KUKA KRL program: MyProgram_168().src

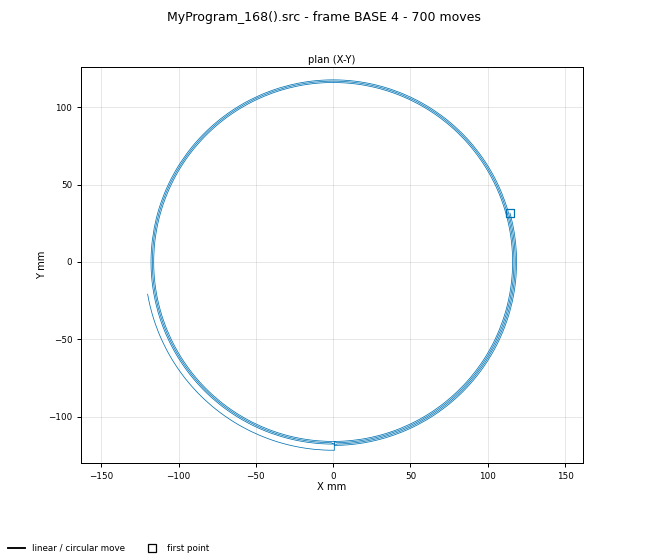
[picture p0: tool path of MyProgram_168().src in frame BASE 4, 700 of 700 moves have a stored position in this frame; points joined in program order, loops and branches not executed]
&ACCESS RVP
&REL 1
&PARAM TEMPLATE = C:\KRC\Roboter\Template\vorgabe
&PARAM EDITMASK = *
DEF MyProgram_168()
; ---- Setting reference (Base) ----
$BASE = BASE_DATA[4]

; --------------------------
; ---- Setting tool (TCP) ----
$TOOL = TOOL_DATA[3]
; --------------------------

$VEL.CP = VEL_APROX_PRINT
Startdeposition()
$VEL.CP = VEL_PRINT
LIN {X 114.3697,Y 31.6504,Z 126,A 10.9682,B 24.9468,C -1.6846,E1 25.1544,E2 435.1117} C_DIS
LIN {X 115.2864,Y 28.1194,Z 126,A 9.3071,B 24.9468,C -1.6839,E1 25.1555,E2 436.7647} C_DIS
LIN {X 116.1642,Y 24.242,Z 126,A 7.4646,B 24.947,C -1.6816,E1 25.1566,E2 438.602} C_DIS
LIN {X 116.7128,Y 21.447,Z 126,A 6.0097,B 24.9475,C -1.6734,E1 25.1574,E2 440.0678} C_DIS
LIN {X 117.2786,Y 18.0937,Z 126,A 4.4449,B 24.9476,C -1.6719,E1 25.1581,E2 441.6268} C_DIS
LIN {X 117.7204,Y 14.9551,Z 126,A 2.982,B 24.9477,C -1.6702,E1 25.1586,E2 443.0851} C_DIS
LIN {X 118.1031,Y 11.5648,Z 126,A 1.1366,B 24.9487,C -1.6553,E1 25.1592,E2 444.9547} C_DIS
LIN {X 118.5333,Y 5.6393,Z 126,A -1.9787,B 24.95,C -1.6341,E1 25.1597,E2 448.1015} C_DIS
LIN {X 118.6444,Y 2.2744,Z 126,A -3.2425,B 24.9492,C -1.6463,E1 25.1597,E2 449.3291} C_DIS
LIN {X 118.6544,Y -1.7308,Z 126,A -5.1222,B 24.9494,C -1.6426,E1 25.1597,E2 451.2063} C_DIS
LIN {X 118.3168,Y -9.105,Z 126,A -8.6006,B 24.9499,C -1.635,E1 25.1593,E2 454.6818} C_DIS
LIN {X 118.0451,Y -12.1269,Z 126,A -10.0562,B 24.9502,C -1.6307,E1 25.1589,E2 456.139} C_DIS
LIN {X 117.691,Y -15.182,Z 126,A -11.6024,B 24.9506,C -1.6229,E1 25.1583,E2 457.6945} C_DIS
LIN {X 117.1469,Y -18.9382,Z 126,A -13.4854,B 24.9512,C -1.6144,E1 25.1575,E2 459.5865} C_DIS
LIN {X 116.5226,Y -22.453,Z 126,A -15.1525,B 24.9513,C -1.6116,E1 25.1567,E2 461.2505} C_DIS
LIN {X 115.7438,Y -26.1788,Z 126,A -16.9413,B 24.9516,C -1.608,E1 25.1556,E2 463.0374} C_DIS
LIN {X 114.3078,Y -31.8689,Z 126,A -19.8139,B 24.9522,C -1.5969,E1 25.1536,E2 465.9193} C_DIS
LIN {X 113.3954,Y -34.9736,Z 126,A -21.3368,B 24.9524,C -1.5939,E1 25.1524,E2 467.4408} C_DIS
LIN {X 112.2692,Y -38.4394,Z 126,A -23.1908,B 24.953,C -1.5837,E1 25.1507,E2 469.3084} C_DIS
LIN {X 110.9509,Y -42.0898,Z 126,A -24.8724,B 24.9528,C -1.5872,E1 25.1491,E2 470.9724} C_DIS
LIN {X 109.7246,Y -45.1929,Z 126,A -27.2104,B 24.9552,C -1.5471,E1 25.1466,E2 473.392} C_DIS
LIN {X 107.7996,Y -49.6101,Z 126,A -28.9531,B 24.9539,C -1.568,E1 25.1446,E2 475.0759} C_DIS
LIN {X 105.9977,Y -53.3542,Z 126,A -30.9386,B 24.9542,C -1.5629,E1 25.1422,E2 477.0628} C_DIS
LIN {X 104.0576,Y -57.0433,Z 126,A -33.1637,B 24.9552,C -1.5467,E1 25.1392,E2 479.3145} C_DIS
LIN {X 102.4696,Y -59.8499,Z 126,A -34.2864,B 24.9542,C -1.563,E1 25.1377,E2 480.3929} C_DIS
LIN {X 99.8547,Y -64.1146,Z 126,A -36.7516,B 24.9548,C -1.5536,E1 25.134,E2 482.8677} C_DIS
LIN {X 96.6923,Y -68.7916,Z 126,A -39.4176,B 24.9551,C -1.5488,E1 25.1298,E2 485.5319} C_DIS
LIN {X 95.1595,Y -70.898,Z 126,A -40.5832,B 24.9551,C -1.5497,E1 25.1279,E2 486.6897} C_DIS
LIN {X 93.2172,Y -73.4318,Z 126,A -42.2808,B 24.9557,C -1.538,E1 25.125,E2 488.4069} C_DIS
LIN {X 91.3145,Y -75.7847,Z 126,A -43.6904,B 24.9557,C -1.5366,E1 25.1225,E2 489.8134} C_DIS
LIN {X 88.1909,Y -79.3985,Z 126,A -46.5348,B 24.9576,C -1.5049,E1 25.1171,E2 492.7198} C_DIS
LIN {X 85.4562,Y -82.334,Z 126,A -47.9476,B 24.9564,C -1.525,E1 25.1145,E2 494.0791} C_DIS
LIN {X 82.8163,Y -84.9914,Z 126,A -49.6649,B 24.9564,C -1.5249,E1 25.1111,E2 495.7894} C_DIS
LIN {X 79.5748,Y -88.0331,Z 126,A -52.338,B 24.9581,C -1.4947,E1 25.1055,E2 498.5229} C_DIS
LIN {X 76.7943,Y -90.4673,Z 126,A -53.6913,B 24.9572,C -1.511,E1 25.1027,E2 499.8323} C_DIS
LIN {X 74.8365,Y -92.0933,Z 126,A -55.2646,B 24.9583,C -1.4919,E1 25.0992,E2 501.4448} C_DIS
LIN {X 72.1024,Y -94.25,Z 126,A -56.6825,B 24.9578,C -1.5007,E1 25.0961,E2 502.8367} C_DIS
LIN {X 68.1758,Y -97.1288,Z 126,A -59.0742,B 24.9582,C -1.4939,E1 25.0907,E2 505.2363} C_DIS
LIN {X 64.6369,Y -99.5195,Z 126,A -60.9796,B 24.958,C -1.4971,E1 25.0863,E2 507.1276} C_DIS
LIN {X 60.6731,Y -101.9831,Z 126,A -63.4892,B 24.9589,C -1.4808,E1 25.0802,E2 509.6679} C_DIS
LIN {X 54.3848,Y -105.471,Z 126,A -66.7011,B 24.9586,C -1.4869,E1 25.0724,E2 512.8561} C_DIS
LIN {X 51.0641,Y -107.1179,Z 126,A -68.4534,B 24.9586,C -1.4858,E1 25.068,E2 514.6065} C_DIS
LIN {X 47.6984,Y -108.6582,Z 126,A -70.2276,B 24.9588,C -1.4836,E1 25.0635,E2 516.3814} C_DIS
LIN {X 44.6734,Y -109.9361,Z 126,A -71.7324,B 24.9587,C -1.4851,E1 25.0596,E2 517.8793} C_DIS
LIN {X 39.1204,Y -112.0325,Z 126,A -75.4311,B 24.961,C -1.4426,E1 25.0497,E2 521.6707} C_DIS
LIN {X 34.1182,Y -113.6563,Z 126,A -77.1593,B 24.9591,C -1.4771,E1 25.0453,E2 523.3144} C_DIS
LIN {X 30.8691,Y -114.5808,Z 126,A -78.7794,B 24.9591,C -1.4758,E1 25.0409,E2 524.9348} C_DIS
LIN {X 27.3135,Y -115.4816,Z 126,A -80.6712,B 24.9596,C -1.4684,E1 25.0358,E2 526.8414} C_DIS
LIN {X 23.5969,Y -116.2967,Z 126,A -82.5163,B 24.9597,C -1.4664,E1 25.0307,E2 528.6889} C_DIS
LIN {X 19.533,Y -117.0475,Z 126,A -84.4332,B 24.9597,C -1.4684,E1 25.0255,E2 530.5989} C_DIS
LIN {X 15.4881,Y -117.6513,Z 126,A -86.4265,B 24.9597,C -1.4662,E1 25.0199,E2 532.5957} C_DIS
LIN {X 11.8786,Y -118.0711,Z 126,A -88.2484,B 24.96,C -1.4621,E1 25.0149,E2 534.4261} C_DIS
LIN {X 9.1459,Y -118.3136,Z 126,A -89.9191,B 24.9608,C -1.4457,E1 25.0101,E2 536.1348} C_DIS
LIN {X 5.3614,Y -118.5453,Z 126,A -91.4312,B 24.9601,C -1.4594,E1 25.006,E2 537.6138} C_DIS
LIN {X 0.8396,Y -118.6625,Z 126,A -93.4659,B 24.9598,C -1.4656,E1 25.0003,E2 539.6336} C_DIS
Enddeposition()
LIN {X 0.8396,Y -118.6625,Z 126,A -93.4659,B 24.9598,C -1.4656,E1 25.0003,E2 539.6336} C_DIS
Startdeposition()
$VEL.CP = VEL_PRINT
LIN {X 2.4206,Y -117.7818,Z 126,A -91.9296,B 24.9569,C -1.5159,E1 25.005,E2 537.9784} C_DIS
LIN {X 6.4049,Y -117.6322,Z 126,A -89.7809,B 24.9564,C -1.5263,E1 25.011,E2 535.8057} C_DIS
LIN {X 10.8382,Y -117.3068,Z 126,A -87.8825,B 24.957,C -1.5152,E1 25.0162,E2 533.9346} C_DIS
LIN {X 14.6658,Y -116.891,Z 126,A -85.9864,B 24.9569,C -1.5174,E1 25.0215,E2 532.0347} C_DIS
LIN {X 18.1381,Y -116.4018,Z 126,A -84.3047,B 24.9569,C -1.5175,E1 25.0261,E2 530.3541} C_DIS
LIN {X 22.0674,Y -115.7213,Z 126,A -82.4187,B 24.9569,C -1.5166,E1 25.0313,E2 528.4724} C_DIS
LIN {X 25.3173,Y -115.0541,Z 126,A -80.7776,B 24.9568,C -1.5194,E1 25.0358,E2 526.827} C_DIS
LIN {X 28.9473,Y -114.1953,Z 126,A -79.1626,B 24.9572,C -1.5119,E1 25.0401,E2 525.232} C_DIS
LIN {X 31.8472,Y -113.4204,Z 126,A -77.4851,B 24.9565,C -1.5236,E1 25.0447,E2 523.5294} C_DIS
LIN {X 37.0934,Y -111.8154,Z 126,A -74.5375,B 24.9556,C -1.54,E1 25.0526,E2 520.5486} C_DIS
LIN {X 42.8622,Y -109.7326,Z 126,A -71.9126,B 24.9563,C -1.5272,E1 25.0594,E2 517.9596} C_DIS
LIN {X 45.9612,Y -108.4711,Z 126,A -70.1681,B 24.9559,C -1.5351,E1 25.064,E2 516.2004} C_DIS
LIN {X 49.2111,Y -107.037,Z 126,A -68.6555,B 24.9563,C -1.5276,E1 25.0677,E2 514.7093} C_DIS
LIN {X 51.8972,Y -105.7604,Z 126,A -67.0473,B 24.9557,C -1.5376,E1 25.0718,E2 513.0816} C_DIS
LIN {X 55.7956,Y -103.7564,Z 126,A -64.1158,B 24.9533,C -1.5795,E1 25.0793,E2 510.0594} C_DIS
LIN {X 60.6656,Y -100.9871,Z 126,A -62.0172,B 24.9547,C -1.5545,E1 25.0842,E2 508.0263} C_DIS
LIN {X 64.6479,Y -98.4838,Z 126,A -59.9825,B 24.9552,C -1.5469,E1 25.0889,E2 506.0161} C_DIS
LIN {X 67.921,Y -96.2564,Z 126,A -58.1836,B 24.9552,C -1.5448,E1 25.093,E2 504.2283} C_DIS
LIN {X 70.3592,Y -94.4881,Z 126,A -55.8829,B 24.9527,C -1.5881,E1 25.0984,E2 501.8337} C_DIS
LIN {X 74.26,Y -91.4539,Z 126,A -54.1692,B 24.9544,C -1.5602,E1 25.1019,E2 500.1923} C_DIS
LIN {X 77.2758,Y -88.9207,Z 126,A -52.1841,B 24.9539,C -1.5679,E1 25.1062,E2 498.1967} C_DIS
LIN {X 81.268,Y -85.2896,Z 126,A -49.5938,B 24.9537,C -1.5725,E1 25.1115,E2 495.6062} C_DIS
LIN {X 83.8102,Y -82.7901,Z 126,A -47.9485,B 24.9537,C -1.5725,E1 25.1147,E2 493.9677} C_DIS
LIN {X 85.8028,Y -80.7231,Z 126,A -46.3875,B 24.953,C -1.584,E1 25.1177,E2 492.3864} C_DIS
LIN {X 88.9954,Y -77.1903,Z 126,A -44.0717,B 24.9526,C -1.5901,E1 25.122,E2 490.0668} C_DIS
LIN {X 91.7991,Y -73.8341,Z 126,A -42.1423,B 24.9529,C -1.5862,E1 25.1254,E2 488.1555} C_DIS
LIN {X 94.8598,Y -69.8575,Z 126,A -39.9365,B 24.9531,C -1.5815,E1 25.1291,E2 485.9711} C_DIS
LIN {X 96.123,Y -68.1092,Z 126,A -38.2088,B 24.951,C -1.6174,E1 25.132,E2 484.1673} C_DIS
LIN {X 98.2882,Y -64.9446,Z 126,A -36.8698,B 24.9522,C -1.5971,E1 25.134,E2 482.8828} C_DIS
LIN {X 100.9275,Y -60.7637,Z 126,A -34.337,B 24.9514,C -1.6103,E1 25.1378,E2 480.3318} C_DIS
LIN {X 104.3384,Y -54.6984,Z 126,A -31.018,B 24.951,C -1.6171,E1 25.1422,E2 477.014} C_DIS
LIN {X 106.4657,Y -50.4342,Z 126,A -28.8487,B 24.951,C -1.6169,E1 25.1449,E2 474.8568} C_DIS
LIN {X 108.9607,Y -44.7893,Z 126,A -25.8268,B 24.9504,C -1.6271,E1 25.1483,E2 471.8273} C_DIS
LIN {X 110.1387,Y -41.807,Z 126,A -24.2461,B 24.95,C -1.633,E1 25.1498,E2 470.2414} C_DIS
LIN {X 111.2128,Y -38.8598,Z 126,A -22.7312,B 24.9498,C -1.6373,E1 25.1513,E2 468.7249} C_DIS
LIN {X 112.4299,Y -35.1849,Z 126,A -20.85,B 24.9494,C -1.6432,E1 25.1529,E2 466.8404} C_DIS
LIN {X 113.6168,Y -31.1392,Z 126,A -18.4461,B 24.9479,C -1.6671,E1 25.1547,E2 464.394} C_DIS
LIN {X 114.4647,Y -27.86,Z 126,A -17.163,B 24.9487,C -1.6546,E1 25.1556,E2 463.1479} C_DIS
LIN {X 115.3289,Y -24.0358,Z 126,A -15.2405,B 24.9483,C -1.6615,E1 25.1567,E2 461.2202} C_DIS
LIN {X 116.0355,Y -20.3561,Z 126,A -13.3673,B 24.9477,C -1.6699,E1 25.1577,E2 459.3382} C_DIS
LIN {X 116.6151,Y -16.712,Z 126,A -11.6978,B 24.9477,C -1.6697,E1 25.1583,E2 457.6791} C_DIS
LIN {X 117.0908,Y -12.9851,Z 126,A -9.7588,B 24.947,C -1.6811,E1 25.159,E2 455.7247} C_DIS
LIN {X 117.4391,Y -9.2962,Z 126,A -8.2226,B 24.9475,C -1.6741,E1 25.1594,E2 454.2141} C_DIS
LIN {X 117.7306,Y -4.2781,Z 126,A -5.5953,B 24.9464,C -1.6909,E1 25.1597,E2 451.5627} C_DIS
LIN {X 117.8015,Y -1.178,Z 126,A -4.1157,B 24.9462,C -1.6945,E1 25.1597,E2 450.0835} C_DIS
LIN {X 117.7804,Y 2.4993,Z 126,A -2.4732,B 24.9462,C -1.6932,E1 25.1597,E2 448.4538} C_DIS
LIN {X 117.6633,Y 5.8427,Z 126,A -0.5556,B 24.945,C -1.7126,E1 25.1595,E2 446.5018} C_DIS
LIN {X 117.3552,Y 10.3138,Z 126,A 1.4516,B 24.9451,C -1.7113,E1 25.159,E2 444.5096} C_DIS
LIN {X 117.0826,Y 13.0552,Z 126,A 2.8311,B 24.9447,C -1.7175,E1 25.1586,E2 443.1236} C_DIS
LIN {X 116.6444,Y 16.5055,Z 126,A 4.4198,B 24.9447,C -1.718,E1 25.158,E2 441.5432} C_DIS
LIN {X 116.0364,Y 20.3509,Z 126,A 6.2799,B 24.9444,C -1.7224,E1 25.1572,E2 439.6837} C_DIS
LIN {X 115.397,Y 23.7043,Z 126,A 7.9493,B 24.944,C -1.7281,E1 25.1563,E2 438.0105} C_DIS
LIN {X 114.5509,Y 27.5069,Z 126,A 9.8717,B 24.9436,C -1.7354,E1 25.1551,E2 436.0821} C_DIS
LIN {X 113.5412,Y 31.4211,Z 126,A 12.2209,B 24.9419,C -1.7601,E1 25.1533,E2 433.6881} C_DIS
LIN {X 112.5143,Y 34.9127,Z 126,A 13.998,B 24.9416,C -1.7659,E1 25.1518,E2 431.9074} C_DIS
LIN {X 111.2946,Y 38.6268,Z 126,A 16.4002,B 24.9395,C -1.7961,E1 25.1495,E2 429.4474} C_DIS
LIN {X 109.1092,Y 44.4245,Z 126,A 18.4351,B 24.9421,C -1.7573,E1 25.1476,E2 427.5152} C_DIS
LIN {X 107.5726,Y 48.0276,Z 126,A 20.3228,B 24.9418,C -1.762,E1 25.1454,E2 425.6269} C_DIS
LIN {X 106.179,Y 51.0331,Z 126,A 21.874,B 24.9417,C -1.7638,E1 25.1436,E2 424.0799} C_DIS
LIN {X 104.4967,Y 54.3977,Z 126,A 23.6806,B 24.9414,C -1.7678,E1 25.1413,E2 422.2734} C_DIS
LIN {X 102.9823,Y 57.2107,Z 126,A 25.717,B 24.9396,C -1.7954,E1 25.1385,E2 420.1826} C_DIS
LIN {X 101.0459,Y 60.569,Z 126,A 27.2329,B 24.9404,C -1.7826,E1 25.1364,E2 418.7046} C_DIS
LIN {X 99.2031,Y 63.5383,Z 126,A 28.8121,B 24.9405,C -1.7814,E1 25.134,E2 417.1362} C_DIS
LIN {X 96.9718,Y 66.8954,Z 126,A 31.4169,B 24.9381,C -1.8174,E1 25.1298,E2 414.4592} C_DIS
LIN {X 94.2992,Y 70.6119,Z 126,A 34.007,B 24.9365,C -1.8405,E1 25.1254,E2 411.8269} C_DIS
LIN {X 90.3594,Y 75.5889,Z 126,A 36.1451,B 24.9391,C -1.8023,E1 25.1218,E2 409.7891} C_DIS
LIN {X 87.8761,Y 78.4613,Z 126,A 37.8874,B 24.9391,C -1.8016,E1 25.1186,E2 408.0561} C_DIS
LIN {X 85.7154,Y 80.8161,Z 126,A 39.4247,B 24.939,C -1.8043,E1 25.1157,E2 406.5192} C_DIS
LIN {X 82.8263,Y 83.7745,Z 126,A 41.4172,B 24.9387,C -1.8078,E1 25.1117,E2 404.5269} C_DIS
LIN {X 80.6047,Y 85.9142,Z 126,A 42.9313,B 24.9385,C -1.8116,E1 25.1087,E2 403.01} C_DIS
LIN {X 78.6641,Y 87.6945,Z 126,A 44.3505,B 24.9379,C -1.8207,E1 25.1057,E2 401.575} C_DIS
LIN {X 75.4647,Y 90.4626,Z 126,A 46.2664,B 24.938,C -1.8181,E1 25.1016,E2 399.6728} C_DIS
LIN {X 73.33,Y 92.2019,Z 126,A 48.1726,B 24.936,C -1.8473,E1 25.0974,E2 397.7046} C_DIS
LIN {X 69.919,Y 94.8148,Z 126,A 49.4916,B 24.9383,C -1.8148,E1 25.0946,E2 396.4672} C_DIS
LIN {X 64.3512,Y 98.6795,Z 126,A 53.0603,B 24.937,C -1.833,E1 25.0863,E2 392.8676} C_DIS
LIN {X 61.2525,Y 100.6305,Z 126,A 54.8975,B 24.9367,C -1.8384,E1 25.0819,E2 391.0235} C_DIS
LIN {X 57.511,Y 102.8146,Z 126,A 56.8262,B 24.937,C -1.8331,E1 25.0773,E2 389.113} C_DIS
LIN {X 54.4099,Y 104.4903,Z 126,A 58.651,B 24.9365,C -1.8405,E1 25.0727,E2 387.2758} C_DIS
LIN {X 50.3531,Y 106.5035,Z 126,A 60.9732,B 24.9359,C -1.8488,E1 25.0669,E2 384.9401} C_DIS
LIN {X 45.9262,Y 108.4858,Z 126,A 62.9554,B 24.9369,C -1.8341,E1 25.0619,E2 382.9976} C_DIS
LIN {X 43.0255,Y 109.6684,Z 126,A 64.6199,B 24.9364,C -1.8421,E1 25.0575,E2 381.3178} C_DIS
LIN {X 36.9847,Y 111.8524,Z 126,A 68.5647,B 24.9336,C -1.8827,E1 25.0469,E2 377.2848} C_DIS
LIN {X 31.8666,Y 113.4149,Z 126,A 70.464,B 24.9357,C -1.8522,E1 25.042,E2 375.4609} C_DIS
LIN {X 28.0302,Y 114.4232,Z 126,A 72.2634,B 24.936,C -1.8475,E1 25.0372,E2 373.6754} C_DIS
LIN {X 24.898,Y 115.1455,Z 126,A 73.8448,B 24.936,C -1.8491,E1 25.0328,E2 372.0923} C_DIS
LIN {X 21.1038,Y 115.901,Z 126,A 75.6984,B 24.936,C -1.8486,E1 25.0278,E2 370.242} C_DIS
LIN {X 17.8305,Y 116.4494,Z 126,A 77.3462,B 24.9358,C -1.8507,E1 25.0232,E2 368.591} C_DIS
LIN {X 14.0522,Y 116.9659,Z 126,A 78.9622,B 24.9365,C -1.8403,E1 25.0188,E2 367.0008} C_DIS
LIN {X 10.606,Y 117.3282,Z 126,A 80.8613,B 24.9358,C -1.8501,E1 25.0135,E2 365.0797} C_DIS
LIN {X 6.8569,Y 117.6072,Z 126,A 82.7423,B 24.9357,C -1.8525,E1 25.0082,E2 363.1937} C_DIS
LIN {X 3.2215,Y 117.763,Z 126,A 84.3745,B 24.9361,C -1.8462,E1 25.0037,E2 361.5769} C_DIS
LIN {X -0.5226,Y 117.8054,Z 126,A 86.2927,B 24.9358,C -1.8502,E1 24.9983,E2 359.6494} C_DIS
LIN {X -4.0567,Y 117.7374,Z 126,A 88.0373,B 24.9358,C -1.8509,E1 24.9935,E2 357.903} C_DIS
LIN {X -7.7851,Y 117.549,Z 126,A 89.8604,B 24.9358,C -1.8505,E1 24.9884,E2 356.0802} C_DIS
LIN {X -11.8034,Y 117.2145,Z 126,A 91.8301,B 24.9358,C -1.8499,E1 24.9829,E2 354.1109} C_DIS
LIN {X -15.3526,Y 116.802,Z 126,A 93.5672,B 24.9359,C -1.8489,E1 24.9781,E2 352.3751} C_DIS
LIN {X -19.1763,Y 116.2355,Z 126,A 95.426,B 24.9361,C -1.8466,E1 24.973,E2 350.52} C_DIS
LIN {X -22.7273,Y 115.5943,Z 126,A 97.2441,B 24.936,C -1.848,E1 24.968,E2 348.6968} C_DIS
LIN {X -27.3774,Y 114.5818,Z 126,A 99.6031,B 24.936,C -1.8478,E1 24.9615,E2 346.3351} C_DIS
LIN {X -34.3237,Y 112.696,Z 126,A 103.1865,B 24.936,C -1.8476,E1 24.9519,E2 342.7464} C_DIS
LIN {X -37.9593,Y 111.5238,Z 126,A 106.0131,B 24.9332,C -1.8879,E1 24.9442,E2 339.8185} C_DIS
LIN {X -44.4418,Y 109.1021,Z 126,A 108.2158,B 24.9371,C -1.8323,E1 24.9388,E2 337.7434} C_DIS
LIN {X -47.6233,Y 107.7531,Z 126,A 110.0371,B 24.9368,C -1.8359,E1 24.9341,E2 335.9093} C_DIS
LIN {X -53.9732,Y 104.7159,Z 126,A 113.3788,B 24.9374,C -1.8268,E1 24.9257,E2 332.5803} C_DIS
LIN {X -57.321,Y 102.9207,Z 126,A 115.2218,B 24.9377,C -1.8234,E1 24.9212,E2 330.7402} C_DIS
LIN {X -60.7272,Y 100.9497,Z 126,A 117.6463,B 24.9364,C -1.8418,E1 24.9153,E2 328.2645} C_DIS
LIN {X -64.161,Y 98.8034,Z 126,A 119.204,B 24.9379,C -1.8203,E1 24.9117,E2 326.753} C_DIS
LIN {X -67.9667,Y 96.2247,Z 126,A 122.1555,B 24.9361,C -1.8466,E1 24.9048,E2 323.7289} C_DIS
LIN {X -72.216,Y 93.0772,Z 126,A 123.7918,B 24.9392,C -1.801,E1 24.9014,E2 322.1951} C_DIS
LIN {X -74.8482,Y 90.9749,Z 126,A 125.6375,B 24.9389,C -1.8061,E1 24.8974,E2 320.3302} C_DIS
LIN {X -79.1923,Y 87.2199,Z 126,A 128.4779,B 24.9392,C -1.8017,E1 24.8914,E2 317.4891} C_DIS
LIN {X -81.4161,Y 85.1469,Z 126,A 130.1934,B 24.9387,C -1.8082,E1 24.8879,E2 315.751} C_DIS
LIN {X -84.7596,Y 81.818,Z 126,A 132.014,B 24.9404,C -1.7826,E1 24.8844,E2 313.9838} C_DIS
LIN {X -87.5458,Y 78.8303,Z 126,A 134.1679,B 24.9404,C -1.7845,E1 24.8803,E2 311.8157} C_DIS
LIN {X -89.7181,Y 76.348,Z 126,A 136.1542,B 24.9395,C -1.7965,E1 24.8767,E2 309.7918} C_DIS
LIN {X -91.8923,Y 73.719,Z 126,A 137.408,B 24.941,C -1.775,E1 24.8745,E2 308.5835} C_DIS
LIN {X -94.3264,Y 70.5758,Z 126,A 139.489,B 24.9409,C -1.7759,E1 24.871,E2 306.4903} C_DIS
LIN {X -98.7986,Y 64.1684,Z 126,A 143.2107,B 24.9418,C -1.7619,E1 24.8651,E2 302.7836} C_DIS
LIN {X -100.386,Y 61.6541,Z 126,A 145.0878,B 24.9409,C -1.7758,E1 24.8623,E2 300.8637} C_DIS
LIN {X -102.1368,Y 58.7062,Z 126,A 146.385,B 24.9422,C -1.7554,E1 24.8606,E2 299.6084} C_DIS
LIN {X -104.584,Y 54.2312,Z 126,A 149.0036,B 24.9424,C -1.7538,E1 24.8571,E2 296.9799} C_DIS
LIN {X -106.2864,Y 50.8096,Z 126,A 150.7093,B 24.9431,C -1.7418,E1 24.855,E2 295.2935} C_DIS
LIN {X -107.8743,Y 47.3452,Z 126,A 152.6246,B 24.9433,C -1.7387,E1 24.8528,E2 293.375} C_DIS
LIN {X -109.183,Y 44.2433,Z 126,A 154.2009,B 24.9438,C -1.7311,E1 24.8512,E2 291.808} C_DIS
LIN {X -111.2638,Y 38.7145,Z 126,A 157.2602,B 24.9439,C -1.7298,E1 24.8482,E2 288.7345} C_DIS
LIN {X -112.4807,Y 35.021,Z 126,A 159.0427,B 24.9446,C -1.7193,E1 24.8467,E2 286.967} C_DIS
LIN {X -113.4229,Y 31.8383,Z 126,A 161.0426,B 24.9439,C -1.7302,E1 24.8452,E2 284.9294} C_DIS
LIN {X -114.3074,Y 28.505,Z 126,A 162.37,B 24.9452,C -1.7102,E1 24.8443,E2 283.6419} C_DIS
LIN {X -115.7358,Y 21.9924,Z 126,A 165.6037,B 24.9459,C -1.6993,E1 24.8424,E2 280.4151} C_DIS
LIN {X -117.0234,Y 13.5611,Z 126,A 169.8068,B 24.9466,C -1.688,E1 24.8407,E2 276.214} C_DIS
LIN {X -117.4027,Y 9.7511,Z 126,A 171.6897,B 24.9469,C -1.6828,E1 24.8402,E2 274.3323} C_DIS
LIN {X -117.6266,Y 6.5073,Z 126,A 173.2935,B 24.9472,C -1.6786,E1 24.84,E2 272.7289} C_DIS
LIN {X -117.7814,Y 2.4448,Z 126,A 175.2773,B 24.9476,C -1.6724,E1 24.8398,E2 270.748} C_DIS
LIN {X -117.8027,Y -0.9985,Z 126,A 177.0597,B 24.9476,C -1.6714,E1 24.8398,E2 268.9571} C_DIS
LIN {X -117.7046,Y -4.9003,Z 126,A 178.8963,B 24.9482,C -1.6626,E1 24.84,E2 267.1302} C_DIS
LIN {X -117.4783,Y -8.8053,Z 126,A -179.1696,B 24.9485,C -1.6578,E1 24.8403,E2 265.1961} C_DIS
LIN {X -117.1632,Y -12.2943,Z 126,A -177.5008,B 24.9489,C -1.6509,E1 24.8408,E2 263.5338} C_DIS
LIN {X -116.7489,Y -15.7621,Z 126,A -175.221,B 24.9478,C -1.6697,E1 24.8417,E2 261.1954} C_DIS
LIN {X -116.1001,Y -19.9863,Z 126,A -173.4496,B 24.949,C -1.6502,E1 24.8425,E2 259.46} C_DIS
LIN {X -114.8936,Y -26.0396,Z 126,A -169.5694,B 24.9472,C -1.678,E1 24.8449,E2 255.4908} C_DIS
LIN {X -113.2243,Y -32.5394,Z 126,A -167.0908,B 24.9499,C -1.6345,E1 24.8467,E2 253.1013} C_DIS
LIN {X -111.7792,Y -37.2019,Z 126,A -164.9393,B 24.9509,C -1.618,E1 24.8485,E2 250.9771} C_DIS
LIN {X -110.5376,Y -40.7424,Z 126,A -163.1418,B 24.9513,C -1.6114,E1 24.8502,E2 249.1851} C_DIS
LIN {X -109.1983,Y -44.2055,Z 126,A -161.3591,B 24.9517,C -1.6051,E1 24.852,E2 247.4075} C_DIS
LIN {X -108.1269,Y -46.7658,Z 126,A -159.1996,B 24.9499,C -1.6355,E1 24.8545,E2 245.1636} C_DIS
LIN {X -105.8983,Y -51.6173,Z 126,A -157.2795,B 24.9521,C -1.5992,E1 24.8567,E2 243.3194} C_DIS
LIN {X -104.2842,Y -54.8011,Z 126,A -155.1944,B 24.9515,C -1.6092,E1 24.8595,E2 241.1994} C_DIS
LIN {X -102.4708,Y -58.1251,Z 126,A -153.6921,B 24.9526,C -1.5897,E1 24.8615,E2 239.7357} C_DIS
LIN {X -100.6338,Y -61.247,Z 126,A -152.0356,B 24.9532,C -1.5806,E1 24.8638,E2 238.0924} C_DIS
LIN {X -97.689,Y -65.8428,Z 126,A -149.3339,B 24.9535,C -1.5756,E1 24.868,E2 235.389} C_DIS
LIN {X -95.9053,Y -68.4143,Z 126,A -147.8593,B 24.9538,C -1.5697,E1 24.8703,E2 233.9212} C_DIS
LIN {X -94.0336,Y -70.9656,Z 126,A -146.213,B 24.9538,C -1.5705,E1 24.8731,E2 232.2652} C_DIS
LIN {X -91.6899,Y -73.9688,Z 126,A -144.3765,B 24.9541,C -1.5653,E1 24.8763,E2 230.4323} C_DIS
LIN {X -89.649,Y -76.4292,Z 126,A -142.6638,B 24.9539,C -1.5684,E1 24.8794,E2 228.7044} C_DIS
LIN {X -87.1946,Y -79.2199,Z 126,A -140.8142,B 24.954,C -1.5661,E1 24.8828,E2 226.852} C_DIS
LIN {X -83.9861,Y -82.6121,Z 126,A -139.0008,B 24.9555,C -1.5415,E1 24.8862,E2 225.0895} C_DIS
LIN {X -81.5196,Y -85.0472,Z 126,A -136.7972,B 24.9544,C -1.5602,E1 24.8908,E2 222.832} C_DIS
LIN {X -77.9802,Y -88.3055,Z 126,A -134.6204,B 24.9551,C -1.5484,E1 24.8952,E2 220.6747} C_DIS
LIN {X -72.8611,Y -92.5725,Z 126,A -131.4414,B 24.9556,C -1.5395,E1 24.9021,E2 217.5046} C_DIS
LIN {X -70.2205,Y -94.5933,Z 126,A -129.3556,B 24.9546,C -1.5571,E1 24.9069,E2 215.3697} C_DIS
LIN {X -67.2508,Y -96.7248,Z 126,A -128.0486,B 24.9559,C -1.5335,E1 24.9097,E2 214.1142} C_DIS
LIN {X -64.2155,Y -98.7684,Z 126,A -126.0418,B 24.9555,C -1.5406,E1 24.9145,E2 212.0841} C_DIS
LIN {X -60.6403,Y -101.0025,Z 126,A -124.2437,B 24.9563,C -1.5264,E1 24.9187,E2 210.314} C_DIS
LIN {X -57.6272,Y -102.7497,Z 126,A -122.4969,B 24.9563,C -1.5264,E1 24.9229,E2 208.5623} C_DIS
LIN {X -53.6019,Y -104.9056,Z 126,A -119.8856,B 24.9555,C -1.5407,E1 24.9295,E2 205.9098} C_DIS
LIN {X -50.4493,Y -106.4595,Z 126,A -118.4359,B 24.9563,C -1.5271,E1 24.9331,E2 204.4887} C_DIS
LIN {X -47.6164,Y -107.7561,Z 126,A -116.8869,B 24.9563,C -1.5269,E1 24.937,E2 202.9364} C_DIS
LIN {X -43.6547,Y -109.4213,Z 126,A -114.4022,B 24.9554,C -1.5424,E1 24.9436,E2 200.4094} C_DIS
LIN {X -39.8251,Y -110.8722,Z 126,A -111.8515,B 24.9541,C -1.5659,E1 24.9505,E2 197.7978} C_DIS
LIN {X -33.5658,Y -112.9234,Z 126,A -109.7511,B 24.9571,C -1.5137,E1 24.9557,E2 195.8176} C_DIS
LIN {X -30.3321,Y -113.8353,Z 126,A -108.0229,B 24.9569,C -1.5169,E1 24.9604,E2 194.0792} C_DIS
LIN {X -26.6052,Y -114.7629,Z 126,A -106.2261,B 24.9571,C -1.5127,E1 24.9653,E2 192.2899} C_DIS
LIN {X -23.1875,Y -115.5031,Z 126,A -104.4205,B 24.9569,C -1.5167,E1 24.9702,E2 190.4728} C_DIS
LIN {X -19.4578,Y -116.1884,Z 126,A -102.6655,B 24.9572,C -1.512,E1 24.975,E2 188.7271} C_DIS
LIN {X -16.1755,Y -116.6913,Z 126,A -100.8062,B 24.9566,C -1.5227,E1 24.9803,E2 186.8409} C_DIS
LIN {X -11.1454,Y -117.2785,Z 126,A -98.6252,B 24.9573,C -1.5096,E1 24.9862,E2 184.6897} C_DIS
LIN {X -7.9671,Y -117.5367,Z 126,A -97.0411,B 24.9573,C -1.5111,E1 24.9907,E2 183.1013} C_DIS
LIN {X -3.7369,Y -117.7472,Z 126,A -94.7479,B 24.9566,C -1.522,E1 24.9971,E2 180.782} C_DIS
LIN {X 0.8282,Y -117.803,Z 126,A -92.8132,B 24.9573,C -1.5094,E1 25.0024,E2 178.8772} C_DIS
Enddeposition()
LIN {X 0.8282,Y -117.803,Z 126,A -92.8132,B 24.9573,C -1.5094,E1 25.0024,E2 178.8772} C_DIS
Startdeposition()
$VEL.CP = VEL_PRINT
LIN {X -1.1886,Y -116.9416,Z 126,A -94.4866,B 24.9582,C -1.4932,E1 24.9977,E2 180.589} C_DIS
LIN {X -4.1628,Y -116.874,Z 126,A -95.9066,B 24.9582,C -1.4946,E1 24.9937,E2 182.0057} C_DIS
LIN {X -7.0084,Y -116.7379,Z 126,A -97.4123,B 24.9584,C -1.4897,E1 24.9895,E2 183.5236} C_DIS
LIN {X -10.832,Y -116.444,Z 126,A -99.1928,B 24.9582,C -1.4941,E1 24.9845,E2 185.2943} C_DIS
LIN {X -13.7897,Y -116.131,Z 126,A -100.7128,B 24.9583,C -1.4915,E1 24.9803,E2 186.8214} C_DIS
LIN {X -17.9645,Y -115.5587,Z 126,A -102.7632,B 24.9583,C -1.4927,E1 24.9746,E2 188.8708} C_DIS
LIN {X -21.8078,Y -114.8958,Z 126,A -104.7402,B 24.9583,C -1.4904,E1 24.9692,E2 190.8552} C_DIS
LIN {X -25.2873,Y -114.1807,Z 126,A -106.4065,B 24.9582,C -1.4944,E1 24.9647,E2 192.514} C_DIS
LIN {X -28.9389,Y -113.3098,Z 126,A -108.2709,B 24.9582,C -1.4944,E1 24.9596,E2 194.3811} C_DIS
LIN {X -32.1543,Y -112.4398,Z 126,A -110.3917,B 24.9593,C -1.4742,E1 24.9538,E2 196.5532} C_DIS
LIN {X -35.8254,Y -111.3243,Z 126,A -111.7737,B 24.958,C -1.4972,E1 24.9502,E2 197.883} C_DIS
LIN {X -38.9017,Y -110.287,Z 126,A -113.4286,B 24.958,C -1.4958,E1 24.9458,E2 199.5446} C_DIS
LIN {X -43.3727,Y -108.6084,Z 126,A -115.723,B 24.9579,C -1.4999,E1 24.9399,E2 201.8339} C_DIS
LIN {X -46.6808,Y -107.2261,Z 126,A -117.4627,B 24.9577,C -1.5026,E1 24.9354,E2 203.5713} C_DIS
LIN {X -49.791,Y -105.8188,Z 126,A -120.357,B 24.9605,C -1.4524,E1 24.9278,E2 206.5921} C_DIS
LIN {X -56.0338,Y -102.6492,Z 126,A -122.0967,B 24.9562,C -1.529,E1 24.9239,E2 208.1545} C_DIS
LIN {X -60.308,Y -100.1985,Z 126,A -125.0963,B 24.9574,C -1.5073,E1 24.9165,E2 211.2148} C_DIS
LIN {X -63.344,Y -98.3063,Z 126,A -126.7308,B 24.957,C -1.5151,E1 24.9127,E2 212.836} C_DIS
LIN {X -66.0351,Y -96.5206,Z 126,A -128.6264,B 24.9576,C -1.5043,E1 24.9082,E2 214.7635} C_DIS
LIN {X -69.7976,Y -93.8357,Z 126,A -130.7925,B 24.9571,C -1.5124,E1 24.9034,E2 216.918} C_DIS
LIN {X -73.1389,Y -91.2559,Z 126,A -132.9458,B 24.9571,C -1.5126,E1 24.8986,E2 219.0787} C_DIS
LIN {X -76.9632,Y -88.0523,Z 126,A -135.186,B 24.9564,C -1.526,E1 24.8939,E2 221.2957} C_DIS
LIN {X -79.9304,Y -85.3682,Z 126,A -137.1646,B 24.9562,C -1.5292,E1 24.8899,E2 223.2747} C_DIS
LIN {X -82.4524,Y -82.9354,Z 126,A -138.7795,B 24.9557,C -1.5371,E1 24.8867,E2 224.8775} C_DIS
LIN {X -84.3696,Y -80.9838,Z 126,A -140.2843,B 24.956,C -1.5332,E1 24.8837,E2 226.3982} C_DIS
LIN {X -86.4067,Y -78.807,Z 126,A -141.6755,B 24.9556,C -1.5394,E1 24.8811,E2 227.7809} C_DIS
LIN {X -89.054,Y -75.8019,Z 126,A -143.6507,B 24.9554,C -1.5434,E1 24.8775,E2 229.7555} C_DIS
LIN {X -91.5092,Y -72.82,Z 126,A -145.7012,B 24.9554,C -1.5413,E1 24.8738,E2 231.8205} C_DIS
LIN {X -94.2327,Y -69.2588,Z 126,A -147.7871,B 24.9549,C -1.5513,E1 24.8704,E2 233.8924} C_DIS
LIN {X -96.4761,Y -66.1008,Z 126,A -149.8121,B 24.9549,C -1.5509,E1 24.8671,E2 235.9285} C_DIS
LIN {X -98.9374,Y -62.355,Z 126,A -151.9374,B 24.9544,C -1.5596,E1 24.8639,E2 238.0438} C_DIS
LIN {X -100.7181,Y -59.434,Z 126,A -153.5529,B 24.954,C -1.5666,E1 24.8616,E2 239.6509} C_DIS
LIN {X -102.5549,Y -56.2076,Z 126,A -155.2554,B 24.9534,C -1.5763,E1 24.8593,E2 241.3391} C_DIS
LIN {X -104.4182,Y -52.6665,Z 126,A -157.4416,B 24.9537,C -1.5725,E1 24.8564,E2 243.5461} C_DIS
LIN {X -106.0066,Y -49.3875,Z 126,A -159.4669,B 24.9539,C -1.5678,E1 24.854,E2 245.5937} C_DIS
LIN {X -107.7505,Y -45.4574,Z 126,A -161.2807,B 24.9529,C -1.5859,E1 24.852,E2 247.3744} C_DIS
LIN {X -109.0688,Y -42.2005,Z 126,A -163.1434,B 24.9529,C -1.5851,E1 24.8501,E2 249.2493} C_DIS
LIN {X -110.3235,Y -38.7978,Z 126,A -164.8337,B 24.9524,C -1.594,E1 24.8485,E2 250.9279} C_DIS
LIN {X -111.5419,Y -35.1459,Z 126,A -166.8379,B 24.9524,C -1.5949,E1 24.8468,E2 252.9415} C_DIS
LIN {X -113.1604,Y -29.52,Z 126,A -169.4116,B 24.9511,C -1.6158,E1 24.8449,E2 255.4804} C_DIS
LIN {X -114.1955,Y -25.2194,Z 126,A -172.5096,B 24.9529,C -1.5848,E1 24.8429,E2 258.6704} C_DIS
LIN {X -115.1601,Y -20.3668,Z 126,A -173.9754,B 24.9501,C -1.6313,E1 24.8422,E2 260.0341} C_DIS
LIN {X -115.9972,Y -14.8732,Z 126,A -176.5176,B 24.9492,C -1.6473,E1 24.8412,E2 262.5532} C_DIS
LIN {X -116.3473,Y -11.8306,Z 126,A -178.4002,B 24.9498,C -1.6365,E1 24.8405,E2 264.4729} C_DIS
LIN {X -116.6124,Y -8.8493,Z 126,A 179.9416,B 24.95,C -1.6334,E1 24.8401,E2 266.1484} C_DIS
LIN {X -116.8351,Y -5.1095,Z 126,A 178.2168,B 24.9494,C -1.6439,E1 24.8399,E2 267.8586} C_DIS
LIN {X -116.9325,Y -1.8477,Z 126,A 176.56,B 24.9492,C -1.6467,E1 24.8398,E2 269.5187} C_DIS
LIN {X -116.9241,Y 2.3071,Z 126,A 174.5398,B 24.9487,C -1.654,E1 24.8398,E2 271.5337} C_DIS
LIN {X -116.8228,Y 5.3944,Z 126,A 173.0153,B 24.9485,C -1.6585,E1 24.84,E2 273.0567} C_DIS
LIN {X -116.6111,Y 8.8658,Z 126,A 171.2568,B 24.9482,C -1.6618,E1 24.8403,E2 274.8177} C_DIS
LIN {X -116.2921,Y 12.3578,Z 126,A 169.066,B 24.9491,C -1.6484,E1 24.841,E2 277.0537} C_DIS
LIN {X -115.8098,Y 16.2684,Z 126,A 167.6094,B 24.9475,C -1.6738,E1 24.8415,E2 278.4586} C_DIS
LIN {X -115.3065,Y 19.5195,Z 126,A 166.0335,B 24.9471,C -1.6805,E1 24.8422,E2 280.0279} C_DIS
LIN {X -114.654,Y 23.0481,Z 126,A 163.949,B 24.9476,C -1.6729,E1 24.8433,E2 282.1425} C_DIS
LIN {X -113.8639,Y 26.6774,Z 126,A 162.3423,B 24.9466,C -1.6874,E1 24.8443,E2 283.7242} C_DIS
LIN {X -112.8396,Y 30.7215,Z 126,A 160.4596,B 24.9458,C -1.7005,E1 24.8456,E2 285.5867} C_DIS
LIN {X -112.035,Y 33.5379,Z 126,A 158.8514,B 24.946,C -1.698,E1 24.8469,E2 287.21} C_DIS
LIN {X -110.8816,Y 37.1732,Z 126,A 156.9926,B 24.9456,C -1.7044,E1 24.8485,E2 289.0644} C_DIS
LIN {X -109.8554,Y 40.1039,Z 126,A 155.3512,B 24.9456,C -1.7043,E1 24.8501,E2 290.7153} C_DIS
LIN {X -108.2239,Y 44.3192,Z 126,A 153.1977,B 24.945,C -1.7136,E1 24.8523,E2 292.8587} C_DIS
LIN {X -106.5681,Y 48.1642,Z 126,A 151.2238,B 24.9444,C -1.723,E1 24.8545,E2 294.821} C_DIS
LIN {X -105.1247,Y 51.2422,Z 126,A 149.5756,B 24.944,C -1.7288,E1 24.8565,E2 296.4644} C_DIS
LIN {X -103.893,Y 53.6943,Z 126,A 148.0457,B 24.9442,C -1.7252,E1 24.8584,E2 298.0108} C_DIS
LIN {X -101.226,Y 58.5659,Z 126,A 145.1872,B 24.9441,C -1.7277,E1 24.8623,E2 300.8786} C_DIS
LIN {X -98.7706,Y 62.6206,Z 126,A 142.971,B 24.9433,C -1.7387,E1 24.8656,E2 303.0799} C_DIS
LIN {X -94.8426,Y 68.4237,Z 126,A 139.698,B 24.9423,C -1.7548,E1 24.8707,E2 306.3307} C_DIS
LIN {X -93.3547,Y 70.4379,Z 126,A 138.3611,B 24.9423,C -1.7537,E1 24.873,E2 307.6767} C_DIS
LIN {X -91.5685,Y 72.745,Z 126,A 136.9302,B 24.9421,C -1.7574,E1 24.8754,E2 309.1053} C_DIS
LIN {X -89.0841,Y 75.7666,Z 126,A 135.0305,B 24.9417,C -1.7632,E1 24.8788,E2 311.0001} C_DIS
LIN {X -86.644,Y 78.5484,Z 126,A 133.0147,B 24.942,C -1.7595,E1 24.8826,E2 313.0338} C_DIS
LIN {X -83.704,Y 81.6743,Z 126,A 130.8877,B 24.9417,C -1.7637,E1 24.8867,E2 315.1599} C_DIS
LIN {X -81.3164,Y 84.049,Z 126,A 129.4195,B 24.9409,C -1.7752,E1 24.8896,E2 316.6068} C_DIS
LIN {X -78.8585,Y 86.3594,Z 126,A 127.779,B 24.9406,C -1.7796,E1 24.893,E2 318.2436} C_DIS
LIN {X -75.8019,Y 89.054,Z 126,A 125.8095,B 24.9403,C -1.7853,E1 24.8971,E2 320.2072} C_DIS
LIN {X -73.2728,Y 91.1474,Z 126,A 124.1948,B 24.94,C -1.7886,E1 24.9006,E2 321.8202} C_DIS
LIN {X -69.0961,Y 94.3518,Z 126,A 121.1326,B 24.941,C -1.774,E1 24.9075,E2 324.9279} C_DIS
LIN {X -66.0932,Y 96.4806,Z 126,A 119.8637,B 24.9393,C -1.7998,E1 24.9103,E2 326.1398} C_DIS
LIN {X -63.0278,Y 98.5092,Z 126,A 117.97,B 24.9393,C -1.7995,E1 24.9148,E2 328.0406} C_DIS
LIN {X -60.4183,Y 100.1314,Z 126,A 116.3915,B 24.9393,C -1.7992,E1 24.9185,E2 329.6245} C_DIS
LIN {X -57.3403,Y 101.9253,Z 126,A 114.6511,B 24.9391,C -1.8026,E1 24.9227,E2 331.3621} C_DIS
LIN {X -54.2763,Y 103.589,Z 126,A 112.9153,B 24.939,C -1.8043,E1 24.927,E2 333.0986} C_DIS
LIN {X -49.9576,Y 105.7413,Z 126,A 110.6676,B 24.9384,C -1.813,E1 24.9326,E2 335.3316} C_DIS
LIN {X -46.3658,Y 107.3634,Z 126,A 108.5874,B 24.9386,C -1.8096,E1 24.938,E2 337.4247} C_DIS
LIN {X -40.9458,Y 109.5456,Z 126,A 105.935,B 24.9377,C -1.8225,E1 24.9448,E2 340.0524} C_DIS
LIN {X -37.2391,Y 110.8594,Z 126,A 103.8691,B 24.938,C -1.819,E1 24.9503,E2 342.1306} C_DIS
LIN {X -29.9906,Y 113.0371,Z 126,A 100.5145,B 24.9367,C -1.8382,E1 24.9592,E2 345.4452} C_DIS
LIN {X -24.4661,Y 114.3598,Z 126,A 97.492,B 24.9372,C -1.8304,E1 24.9674,E2 348.4902} C_DIS
LIN {X -22.0892,Y 114.8417,Z 126,A 96.1681,B 24.9375,C -1.8256,E1 24.9711,E2 349.8271} C_DIS
LIN {X -18.324,Y 115.5032,Z 126,A 94.2691,B 24.9375,C -1.8258,E1 24.9763,E2 351.7274} C_DIS
LIN {X -14.9334,Y 115.9894,Z 126,A 92.6014,B 24.9375,C -1.8274,E1 24.9809,E2 353.3927} C_DIS
LIN {X -11.8802,Y 116.3421,Z 126,A 91.124,B 24.9373,C -1.8294,E1 24.985,E2 354.8661} C_DIS
LIN {X -8.2074,Y 116.6588,Z 126,A 89.2394,B 24.9374,C -1.8268,E1 24.9903,E2 356.7577} C_DIS
LIN {X -4.7436,Y 116.8508,Z 126,A 87.5737,B 24.9374,C -1.8289,E1 24.9949,E2 358.4188} C_DIS
LIN {X -0.8286,Y 116.9438,Z 126,A 85.6311,B 24.9374,C -1.8283,E1 25.0003,E2 360.3629} C_DIS
LIN {X 2.3357,Y 116.9235,Z 126,A 84.14,B 24.9371,C -1.8311,E1 25.0045,E2 361.8471} C_DIS
LIN {X 5.822,Y 116.8034,Z 126,A 82.25,B 24.9377,C -1.8233,E1 25.0098,E2 363.7552} C_DIS
LIN {X 9.8141,Y 116.5353,Z 126,A 80.3918,B 24.9374,C -1.8277,E1 25.0149,E2 365.6021} C_DIS
LIN {X 13.71,Y 116.1404,Z 126,A 78.543,B 24.9372,C -1.8305,E1 25.02,E2 367.443} C_DIS
LIN {X 17.2085,Y 115.6756,Z 126,A 76.7007,B 24.9376,C -1.825,E1 25.0252,E2 369.2966} C_DIS
LIN {X 21.0457,Y 115.038,Z 126,A 74.7671,B 24.9377,C -1.8231,E1 25.0305,E2 371.2327} C_DIS
LIN {X 24.9867,Y 114.2463,Z 126,A 72.9554,B 24.9373,C -1.8291,E1 25.0354,E2 373.0278} C_DIS
LIN {X 28.433,Y 113.4398,Z 126,A 70.6772,B 24.939,C -1.804,E1 25.0417,E2 375.3621} C_DIS
LIN {X 32.2015,Y 112.4265,Z 126,A 69.4546,B 24.937,C -1.8333,E1 25.0448,E2 376.5134} C_DIS
LIN {X 34.7485,Y 111.6651,Z 126,A 67.9988,B 24.9375,C -1.8255,E1 25.0488,E2 377.9852} C_DIS
LIN {X 38.1093,Y 110.5651,Z 126,A 66.02,B 24.9384,C -1.813,E1 25.0541,E2 379.9897} C_DIS
LIN {X 42.1595,Y 109.0849,Z 126,A 64.037,B 24.9381,C -1.8167,E1 25.0592,E2 381.9596} C_DIS
LIN {X 45.6212,Y 107.6814,Z 126,A 62.3412,B 24.9379,C -1.8208,E1 25.0635,E2 383.6418} C_DIS
LIN {X 52.0371,Y 104.7315,Z 126,A 58.8419,B 24.9383,C -1.8148,E1 25.0724,E2 387.1462} C_DIS
LIN {X 55.9218,Y 102.7099,Z 126,A 56.7383,B 24.9383,C -1.8138,E1 25.0776,E2 389.2462} C_DIS
LIN {X 58.7885,Y 101.098,Z 126,A 55.1735,B 24.9383,C -1.8136,E1 25.0814,E2 390.8069} C_DIS
LIN {X 60.9598,Y 99.8023,Z 126,A 53.9559,B 24.9384,C -1.8127,E1 25.0843,E2 392.0228} C_DIS
LIN {X 63.4853,Y 98.2155,Z 126,A 51.9886,B 24.9401,C -1.7874,E1 25.089,E2 394.0436} C_DIS
LIN {X 66.527,Y 96.1809,Z 126,A 50.8944,B 24.9382,C -1.8162,E1 25.0914,E2 395.066} C_DIS
LIN {X 69.9064,Y 93.754,Z 126,A 48.3608,B 24.9399,C -1.79,E1 25.0972,E2 397.6526} C_DIS
LIN {X 73.5519,Y 90.9212,Z 126,A 46.3372,B 24.9395,C -1.7967,E1 25.1016,E2 399.6528} C_DIS
LIN {X 76.5412,Y 88.4209,Z 126,A 44.0534,B 24.9409,C -1.7757,E1 25.1065,E2 401.9773} C_DIS
LIN {X 79.1067,Y 86.1317,Z 126,A 42.8746,B 24.9396,C -1.7955,E1 25.1089,E2 403.1045} C_DIS
LIN {X 81.0249,Y 84.3299,Z 126,A 41.5009,B 24.94,C -1.7889,E1 25.1117,E2 404.4882} C_DIS
LIN {X 85.2605,Y 80.045,Z 126,A 38.5889,B 24.9403,C -1.7843,E1 25.1173,E2 407.3986} C_DIS
LIN {X 87.0404,Y 78.1059,Z 126,A 37.2693,B 24.9406,C -1.7799,E1 25.1198,E2 408.7226} C_DIS
LIN {X 89.4357,Y 75.3538,Z 126,A 34.982,B 24.9424,C -1.7526,E1 25.1241,E2 411.0641} C_DIS
LIN {X 91.9156,Y 72.3058,Z 126,A 33.6104,B 24.941,C -1.7736,E1 25.1263,E2 412.3797} C_DIS
LIN {X 94.1931,Y 69.3129,Z 126,A 31.5248,B 24.9421,C -1.7576,E1 25.1299,E2 414.4929} C_DIS
LIN {X 97.0383,Y 65.2705,Z 126,A 29.3744,B 24.9417,C -1.7641,E1 25.1332,E2 416.6175} C_DIS
LIN {X 98.5957,Y 62.8931,Z 126,A 28.0224,B 24.9417,C -1.7623,E1 25.1353,E2 417.9669} C_DIS
LIN {X 100.3862,Y 59.9956,Z 126,A 25.5437,B 24.9446,C -1.72,E1 25.139,E2 420.5327} C_DIS
LIN {X 102.8747,Y 55.618,Z 126,A 23.8791,B 24.9426,C -1.7507,E1 25.1411,E2 422.1163} C_DIS
LIN {X 104.5955,Y 52.3114,Z 126,A 21.9408,B 24.9432,C -1.7403,E1 25.1436,E2 424.0689} C_DIS
LIN {X 106.2647,Y 48.8332,Z 126,A 20.2144,B 24.9431,C -1.7426,E1 25.1456,E2 425.7806} C_DIS
LIN {X 107.525,Y 45.9923,Z 126,A 18.5396,B 24.9438,C -1.7309,E1 25.1475,E2 427.4737} C_DIS
LIN {X 109.5954,Y 40.8143,Z 126,A 15.7909,B 24.9444,C -1.722,E1 25.1503,E2 430.2281} C_DIS
LIN {X 110.9173,Y 37.0672,Z 126,A 13.9933,B 24.9444,C -1.7232,E1 25.1519,E2 432.0126} C_DIS
LIN {X 112.7126,Y 31.1918,Z 126,A 10.9353,B 24.9451,C -1.7117,E1 25.1544,E2 435.0805} C_DIS
LIN {X 113.5792,Y 27.8626,Z 126,A 9.315,B 24.9452,C -1.7096,E1 25.1555,E2 436.6964} C_DIS
LIN {X 114.3476,Y 24.5223,Z 126,A 7.6426,B 24.9455,C -1.7046,E1 25.1565,E2 438.3709} C_DIS
LIN {X 115.0387,Y 21.0419,Z 126,A 5.8668,B 24.946,C -1.6973,E1 25.1574,E2 440.1534} C_DIS
LIN {X 115.6591,Y 17.3155,Z 126,A 3.9831,B 24.9465,C -1.6898,E1 25.1582,E2 442.0437} C_DIS
LIN {X 116.1822,Y 13.353,Z 126,A 2.0879,B 24.9467,C -1.6865,E1 25.1589,E2 443.9355} C_DIS
LIN {X 116.5662,Y 9.4276,Z 126,A 0.2369,B 24.9468,C -1.6842,E1 25.1593,E2 445.7811} C_DIS
LIN {X 116.791,Y 6.0466,Z 126,A -1.4784,B 24.9474,C -1.6761,E1 25.1596,E2 447.5051} C_DIS
LIN {X 116.9258,Y 2.2154,Z 126,A -3.2661,B 24.9474,C -1.6743,E1 25.1598,E2 449.2865} C_DIS
LIN {X 116.941,Y -1.3005,Z 126,A -4.9769,B 24.9478,C -1.6692,E1 25.1598,E2 450.9991} C_DIS
LIN {X 116.8482,Y -4.8045,Z 126,A -6.8303,B 24.9485,C -1.6571,E1 25.1596,E2 452.8699} C_DIS
LIN {X 116.5995,Y -9.0108,Z 126,A -8.7858,B 24.9486,C -1.6556,E1 25.1592,E2 454.8175} C_DIS
LIN {X 116.2461,Y -12.797,Z 126,A -10.6696,B 24.9491,C -1.6485,E1 25.1587,E2 456.707} C_DIS
LIN {X 115.8106,Y -16.2626,Z 126,A -12.3076,B 24.9492,C -1.6464,E1 25.1581,E2 458.3401} C_DIS
LIN {X 115.3393,Y -19.3231,Z 126,A -13.8018,B 24.9494,C -1.6425,E1 25.1574,E2 459.8346} C_DIS
LIN {X 114.6807,Y -22.9183,Z 126,A -15.6791,B 24.9501,C -1.6326,E1 25.1564,E2 461.7245} C_DIS
LIN {X 113.9303,Y -26.3898,Z 126,A -17.3056,B 24.9501,C -1.6324,E1 25.1554,E2 463.342} C_DIS
LIN {X 112.1294,Y -33.2196,Z 126,A -20.403,B 24.9497,C -1.6386,E1 25.1533,E2 466.4069} C_DIS
LIN {X 110.8558,Y -37.2498,Z 126,A -22.4943,B 24.9502,C -1.631,E1 25.1515,E2 468.5043} C_DIS
LIN {X 109.476,Y -41.1295,Z 126,A -24.8623,B 24.9516,C -1.6079,E1 25.1492,E2 470.9136} C_DIS
LIN {X 108.1993,Y -44.3795,Z 126,A -26.7302,B 24.9523,C -1.595,E1 25.1472,E2 472.8013} C_DIS
LIN {X 105.3053,Y -50.8663,Z 126,A -29.5607,B 24.9511,C -1.6153,E1 25.1441,E2 475.5686} C_DIS
LIN {X 104.1788,Y -53.135,Z 126,A -31.2259,B 24.9526,C -1.5913,E1 25.1419,E2 477.2815} C_DIS
LIN {X 101.5762,Y -57.9563,Z 126,A -33.9119,B 24.953,C -1.5832,E1 25.1383,E2 479.9726} C_DIS
LIN {X 99.8822,Y -60.8285,Z 126,A -35.5003,B 24.9532,C -1.5806,E1 25.136,E2 481.5591} C_DIS
LIN {X 98.359,Y -63.2619,Z 126,A -36.8448,B 24.9532,C -1.5795,E1 25.134,E2 482.8994} C_DIS
LIN {X 95.6203,Y -67.3334,Z 126,A -39.3254,B 24.9539,C -1.5691,E1 25.1301,E2 485.3925} C_DIS
LIN {X 93.0916,Y -70.7881,Z 126,A -41.4549,B 24.9543,C -1.5618,E1 25.1265,E2 487.5289} C_DIS
LIN {X 90.8474,Y -73.643,Z 126,A -43.1836,B 24.9544,C -1.5594,E1 25.1235,E2 489.2552} C_DIS
LIN {X 87.6245,Y -77.453,Z 126,A -45.5119,B 24.9544,C -1.5584,E1 25.1193,E2 491.5751} C_DIS
LIN {X 86.0467,Y -79.1993,Z 126,A -46.6631,B 24.9547,C -1.5556,E1 25.1171,E2 492.7279} C_DIS
LIN {X 83.6606,Y -81.7182,Z 126,A -48.504,B 24.9553,C -1.5446,E1 25.1135,E2 494.5867} C_DIS
LIN {X 81.1022,Y -84.2554,Z 126,A -50.1491,B 24.9553,C -1.546,E1 25.1102,E2 496.2217} C_DIS
LIN {X 78.4392,Y -86.742,Z 126,A -51.8262,B 24.9552,C -1.5468,E1 25.1068,E2 497.8901} C_DIS
LIN {X 76.7795,Y -88.2128,Z 126,A -53.0289,B 24.9556,C -1.5388,E1 25.1043,E2 499.1069} C_DIS
LIN {X 73.6802,Y -90.8172,Z 126,A -55.6682,B 24.9576,C -1.5038,E1 25.0984,E2 501.8188} C_DIS
LIN {X 69.9153,Y -93.7472,Z 126,A -57.273,B 24.956,C -1.5328,E1 25.095,E2 503.3493} C_DIS
LIN {X 66.2085,Y -96.4023,Z 126,A -59.6618,B 24.9567,C -1.5209,E1 25.0895,E2 505.7579} C_DIS
LIN {X 63.1352,Y -98.4402,Z 126,A -61.3382,B 24.9565,C -1.5235,E1 25.0856,E2 507.4228} C_DIS
LIN {X 60.7791,Y -99.9121,Z 126,A -63.274,B 24.9582,C -1.4943,E1 25.0808,E2 509.4215} C_DIS
LIN {X 57.0782,Y -102.0716,Z 126,A -65.3334,B 24.9582,C -1.4923,E1 25.0758,E2 511.4795} C_DIS
LIN {X 53.4199,Y -104.0332,Z 126,A -67.0684,B 24.9577,C -1.5026,E1 25.0716,E2 513.1853} C_DIS
LIN {X 48.7744,Y -106.2919,Z 126,A -69.4043,B 24.9574,C -1.5075,E1 25.0657,E2 515.5037} C_DIS
LIN {X 45.5892,Y -107.6949,Z 126,A -71.0934,B 24.9575,C -1.5057,E1 25.0614,E2 517.1931} C_DIS
LIN {X 42.3224,Y -109.0209,Z 126,A -72.7143,B 24.9574,C -1.5081,E1 25.0572,E2 518.8046} C_DIS
LIN {X 34.8343,Y -111.6385,Z 126,A -76.5263,B 24.9574,C -1.5065,E1 25.0472,E2 522.6128} C_DIS
LIN {X 32.6668,Y -112.2934,Z 126,A -78.0013,B 24.9585,C -1.4885,E1 25.0431,E2 524.1279} C_DIS
LIN {X 27.7702,Y -113.6017,Z 126,A -80.1944,B 24.9579,C -1.4991,E1 25.0373,E2 526.2924} C_DIS
LIN {X 24.2687,Y -114.4029,Z 126,A -82.0689,B 24.9583,C -1.4923,E1 25.0321,E2 528.1807} C_DIS
LIN {X 20.7261,Y -115.0955,Z 126,A -83.738,B 24.9581,C -1.4953,E1 25.0275,E2 529.8407} C_DIS
LIN {X 17.0496,Y -115.6988,Z 126,A -85.6992,B 24.9585,C -1.4878,E1 25.0221,E2 531.8178} C_DIS
LIN {X 13.3112,Y -116.1871,Z 126,A -87.4236,B 24.9583,C -1.4922,E1 25.0173,E2 533.5304} C_DIS
LIN {X 9.4582,Y -116.5637,Z 126,A -89.3581,B 24.9584,C -1.4895,E1 25.0119,E2 535.4703} C_DIS
LIN {X 5.5518,Y -116.8161,Z 126,A -91.2038,B 24.9583,C -1.4919,E1 25.0068,E2 537.3095} C_DIS
LIN {X 2.2136,Y -116.9258,Z 126,A -92.8329,B 24.9583,C -1.4918,E1 25.0023,E2 538.9386} C_DIS
LIN {X 2.2136,Y -116.9258,Z 126,A -92.8329,B 24.9583,C -1.4918,E1 25.0023,E2 538.9386} C_DIS
Enddeposition()
LIN {X 0.8095,Y -116.0815,Z 126,A -93.0674,B 24.9563,C -1.527,E1 25.0019,E2 539.0896} C_DIS
Startdeposition()
$VEL.CP = VEL_PRINT
LIN {X 4.2618,Y -116.0109,Z 126,A -91.005,B 24.9554,C -1.5436,E1 25.0077,E2 536.9883} C_DIS
LIN {X 7.1,Y -115.8718,Z 126,A -89.599,B 24.9554,C -1.5443,E1 25.0116,E2 535.5812} C_DIS
LIN {X 11.378,Y -115.5303,Z 126,A -87.6631,B 24.9557,C -1.5372,E1 25.017,E2 533.6633} C_DIS
LIN {X 14.2044,Y -115.2169,Z 126,A -86.0849,B 24.9552,C -1.546,E1 25.0214,E2 532.0654} C_DIS
LIN {X 17.0219,Y -114.8344,Z 126,A -84.6826,B 24.9552,C -1.5469,E1 25.0253,E2 530.6622} C_DIS
LIN {X 20.5478,Y -114.254,Z 126,A -83.1364,B 24.9557,C -1.5384,E1 25.0295,E2 529.1377} C_DIS
LIN {X 24.0439,Y -113.572,Z 126,A -81.1671,B 24.955,C -1.5496,E1 25.0349,E2 527.1444} C_DIS
LIN {X 27.3604,Y -112.8168,Z 126,A -79.6701,B 24.9554,C -1.5429,E1 25.039,E2 525.6653} C_DIS
LIN {X 31.0318,Y -111.8644,Z 126,A -77.8199,B 24.9554,C -1.5439,E1 25.0439,E2 523.8158} C_DIS
LIN {X 33.972,Y -111.0058,Z 126,A -76.2306,B 24.955,C -1.5492,E1 25.0482,E2 522.2167} C_DIS
LIN {X 36.8206,Y -110.0932,Z 126,A -74.8518,B 24.9552,C -1.5465,E1 25.0519,E2 520.8467} C_DIS
LIN {X 40.005,Y -108.9764,Z 126,A -73.1066,B 24.9548,C -1.5524,E1 25.0565,E2 519.0912} C_DIS
LIN {X 43.5267,Y -107.6183,Z 126,A -71.2743,B 24.9548,C -1.5536,E1 25.0612,E2 517.2601} C_DIS
LIN {X 47.5435,Y -105.9049,Z 126,A -69.3978,B 24.9553,C -1.544,E1 25.066,E2 515.4109} C_DIS
LIN {X 49.6204,Y -104.95,Z 126,A -68.0295,B 24.9546,C -1.5569,E1 25.0695,E2 514.0157} C_DIS
LIN {X 52.6958,Y -103.4378,Z 126,A -66.3487,B 24.9544,C -1.5592,E1 25.0737,E2 512.3339} C_DIS
LIN {X 55.941,Y -101.7214,Z 126,A -64.3765,B 24.9538,C -1.5698,E1 25.0786,E2 510.3422} C_DIS
LIN {X 59.1088,Y -99.9117,Z 126,A -62.6518,B 24.9538,C -1.5696,E1 25.0827,E2 508.6233} C_DIS
LIN {X 62.1075,Y -98.0783,Z 126,A -61.0164,B 24.9539,C -1.5683,E1 25.0866,E2 506.9962} C_DIS
LIN {X 64.9568,Y -96.2124,Z 126,A -59.3364,B 24.9537,C -1.5716,E1 25.0905,E2 505.3139} C_DIS
LIN {X 67.3098,Y -94.5812,Z 126,A -57.9403,B 24.9536,C -1.5738,E1 25.0937,E2 503.9176} C_DIS
LIN {X 69.5901,Y -92.9163,Z 126,A -56.5134,B 24.9533,C -1.5783,E1 25.0969,E2 502.4851} C_DIS
LIN {X 71.9541,Y -91.0978,Z 126,A -55.0746,B 24.9533,C -1.58,E1 25.1001,E2 501.0477} C_DIS
LIN {X 74.1925,Y -89.2842,Z 126,A -53.6697,B 24.9531,C -1.5824,E1 25.1031,E2 499.6425} C_DIS
LIN {X 76.3576,Y -87.4398,Z 126,A -52.273,B 24.9529,C -1.5853,E1 25.1061,E2 498.2443} C_DIS
LIN {X 78.493,Y -85.528,Z 126,A -50.8656,B 24.9527,C -1.5883,E1 25.109,E2 496.8355} C_DIS
LIN {X 80.5642,Y -83.5799,Z 126,A -49.4692,B 24.9526,C -1.5913,E1 25.1118,E2 495.4377} C_DIS
LIN {X 82.5872,Y -81.5815,Z 126,A -48.0732,B 24.9524,C -1.5945,E1 25.1146,E2 494.0403} C_DIS
LIN {X 84.5606,Y -79.5342,Z 126,A -46.6772,B 24.9522,C -1.5976,E1 25.1173,E2 492.6427} C_DIS
LIN {X 86.6671,Y -77.234,Z 126,A -45.1978,B 24.9522,C -1.5988,E1 25.12,E2 491.1672} C_DIS
LIN {X 88.8305,Y -74.7385,Z 126,A -43.4226,B 24.9514,C -1.6099,E1 25.1233,E2 489.3738} C_DIS
LIN {X 90.8069,Y -72.3221,Z 126,A -41.9437,B 24.9514,C -1.6111,E1 25.1259,E2 487.899} C_DIS
LIN {X 92.3834,Y -70.2994,Z 126,A -40.7311,B 24.9514,C -1.612,E1 25.1279,E2 486.6899} C_DIS
LIN {X 94.0836,Y -68.0072,Z 126,A -39.334,B 24.9511,C -1.6154,E1 25.1302,E2 485.2916} C_DIS
LIN {X 95.7121,Y -65.6952,Z 126,A -37.7678,B 24.9504,C -1.6275,E1 25.1327,E2 483.7047} C_DIS
LIN {X 97.6106,Y -62.8362,Z 126,A -36.2525,B 24.9506,C -1.6238,E1 25.135,E2 482.2056} C_DIS
LIN {X 99.1259,Y -60.4175,Z 126,A -34.864,B 24.9504,C -1.6269,E1 25.1371,E2 480.8168} C_DIS
LIN {X 101.1805,Y -56.9108,Z 126,A -32.8049,B 24.9499,C -1.6354,E1 25.14,E2 478.7484} C_DIS
LIN {X 103.1102,Y -53.3367,Z 126,A -30.7517,B 24.9494,C -1.6437,E1 25.1426,E2 476.6865} C_DIS
LIN {X 104.5584,Y -50.4358,Z 126,A -29.2909,B 24.9494,C -1.6419,E1 25.1444,E2 475.2378} C_DIS
LIN {X 106.3271,Y -46.5917,Z 126,A -27.1438,B 24.9489,C -1.6511,E1 25.1469,E2 473.0805} C_DIS
LIN {X 107.5482,Y -43.6988,Z 126,A -25.7264,B 24.949,C -1.6496,E1 25.1484,E2 471.6745} C_DIS
LIN {X 109.0044,Y -39.9283,Z 126,A -23.9364,B 24.9492,C -1.646,E1 25.1502,E2 469.9029} C_DIS
LIN {X 109.7715,Y -37.7745,Z 126,A -22.5702,B 24.9483,C -1.6609,E1 25.1515,E2 468.5093} C_DIS
LIN {X 110.8364,Y -34.5181,Z 126,A -20.8946,B 24.948,C -1.6656,E1 25.1529,E2 466.8321} C_DIS
LIN {X 111.8762,Y -30.9899,Z 126,A -19.0879,B 24.9477,C -1.6709,E1 25.1543,E2 465.0232} C_DIS
LIN {X 112.6112,Y -28.203,Z 126,A -17.6734,B 24.9474,C -1.6751,E1 25.1553,E2 463.607} C_DIS
LIN {X 113.3882,Y -24.8867,Z 126,A -16.0061,B 24.9471,C -1.6799,E1 25.1563,E2 461.9379} C_DIS
LIN {X 114.2273,Y -20.6967,Z 126,A -13.9375,B 24.9468,C -1.6848,E1 25.1574,E2 459.8699} C_DIS
LIN {X 114.8342,Y -17.0235,Z 126,A -11.9104,B 24.9458,C -1.6999,E1 25.1583,E2 457.8192} C_DIS
LIN {X 115.2815,Y -13.6528,Z 126,A -10.4202,B 24.9461,C -1.6964,E1 25.1588,E2 456.346} C_DIS
LIN {X 115.5968,Y -10.6577,Z 126,A -8.9157,B 24.9457,C -1.7021,E1 25.1592,E2 454.8369} C_DIS
LIN {X 115.8703,Y -7.1257,Z 126,A -7.0267,B 24.9449,C -1.7146,E1 25.1596,E2 452.9299} C_DIS
LIN {X 116.0108,Y -4.2653,Z 126,A -5.8045,B 24.9452,C -1.71,E1 25.1597,E2 451.7257} C_DIS
LIN {X 116.0805,Y -1.423,Z 126,A -4.2659,B 24.9445,C -1.7211,E1 25.1597,E2 450.1701} C_DIS
LIN {X 116.0703,Y 1.9769,Z 126,A -2.7442,B 24.9446,C -1.7191,E1 25.1597,E2 448.6621} C_DIS
LIN {X 115.9181,Y 6.2627,Z 126,A -0.8874,B 24.945,C -1.7136,E1 25.1595,E2 446.8294} C_DIS
LIN {X 115.7299,Y 9.0994,Z 126,A 0.7515,B 24.944,C -1.7294,E1 25.1592,E2 445.163} C_DIS
LIN {X 115.3824,Y 12.7908,Z 126,A 2.7353,B 24.9431,C -1.7426,E1 25.1586,E2 443.1597} C_DIS
LIN {X 114.9316,Y 16.3376,Z 126,A 4.3526,B 24.9431,C -1.7413,E1 25.158,E2 441.5552} C_DIS
LIN {X 114.3793,Y 19.8513,Z 126,A 6.2424,B 24.9424,C -1.7532,E1 25.1572,E2 439.6482} C_DIS
LIN {X 113.8588,Y 22.6467,Z 126,A 7.4599,B 24.9427,C -1.7488,E1 25.1565,E2 438.4483} C_DIS
LIN {X 113.145,Y 25.9698,Z 126,A 9.1776,B 24.9422,C -1.756,E1 25.1555,E2 436.7236} C_DIS
LIN {X 112.4697,Y 28.754,Z 126,A 10.5302,B 24.9422,C -1.7575,E1 25.1546,E2 435.3753} C_DIS
LIN {X 111.7076,Y 31.5851,Z 126,A 12.0201,B 24.9417,C -1.764,E1 25.1535,E2 433.8786} C_DIS
LIN {X 110.663,Y 35.0767,Z 126,A 13.9286,B 24.941,C -1.7747,E1 25.1519,E2 431.9557} C_DIS
LIN {X 109.3053,Y 39.103,Z 126,A 16.0133,B 24.9406,C -1.7804,E1 25.15,E2 429.8692} C_DIS
LIN {X 108.3187,Y 41.758,Z 126,A 17.2283,B 24.9409,C -1.7759,E1 25.1488,E2 428.6717} C_DIS
LIN {X 107.1235,Y 44.7314,Z 126,A 18.8824,B 24.9403,C -1.784,E1 25.147,E2 427.0075} C_DIS
LIN {X 105.5439,Y 48.3445,Z 126,A 20.734,B 24.9403,C -1.7851,E1 25.1449,E2 425.1635} C_DIS
LIN {X 104.3282,Y 50.9149,Z 126,A 22.3057,B 24.9395,C -1.7971,E1 25.143,E2 423.5719} C_DIS
LIN {X 102.7773,Y 53.9725,Z 126,A 23.6486,B 24.9403,C -1.7854,E1 25.1413,E2 422.2638} C_DIS
LIN {X 101.7299,Y 55.9255,Z 126,A 25.0408,B 24.9391,C -1.8025,E1 25.1394,E2 420.8385} C_DIS
LIN {X 100.0057,Y 58.9498,Z 126,A 26.5971,B 24.9393,C -1.7995,E1 25.1372,E2 419.2972} C_DIS
LIN {X 98.4813,Y 61.4625,Z 126,A 28.0917,B 24.9389,C -1.8055,E1 25.135,E2 417.7962} C_DIS
LIN {X 96.5256,Y 64.4942,Z 126,A 29.997,B 24.9382,C -1.816,E1 25.1321,E2 415.8756} C_DIS
LIN {X 94.5054,Y 67.4161,Z 126,A 31.5302,B 24.9386,C -1.8101,E1 25.1297,E2 414.3637} C_DIS
LIN {X 92.9086,Y 69.6003,Z 126,A 32.9281,B 24.9382,C -1.8164,E1 25.1273,E2 412.9577} C_DIS
LIN {X 91.0857,Y 71.9694,Z 126,A 34.3581,B 24.9381,C -1.8179,E1 25.1249,E2 411.5309} C_DIS
LIN {X 89.3019,Y 74.1713,Z 126,A 35.7934,B 24.9377,C -1.8229,E1 25.1223,E2 410.0903} C_DIS
LIN {X 86.967,Y 76.8989,Z 126,A 37.6614,B 24.9371,C -1.8315,E1 25.1189,E2 408.2105} C_DIS
LIN {X 84.7555,Y 79.327,Z 126,A 39.1965,B 24.9371,C -1.8312,E1 25.116,E2 406.6828} C_DIS
LIN {X 82.4158,Y 81.7551,Z 126,A 40.7411,B 24.9373,C -1.8293,E1 25.113,E2 405.1493} C_DIS
LIN {X 80.562,Y 83.582,Z 126,A 42.0625,B 24.937,C -1.8337,E1 25.1103,E2 403.823} C_DIS
LIN {X 78.486,Y 85.5345,Z 126,A 43.4606,B 24.9368,C -1.8363,E1 25.1075,E2 402.4246} C_DIS
LIN {X 76.1534,Y 87.6181,Z 126,A 45.1474,B 24.9361,C -1.846,E1 25.1039,E2 400.7216} C_DIS
LIN {X 73.4325,Y 89.9113,Z 126,A 46.7488,B 24.9364,C -1.8422,E1 25.1005,E2 399.1352} C_DIS
LIN {X 71.0861,Y 91.7771,Z 126,A 48.0429,B 24.9368,C -1.8364,E1 25.0977,E2 397.8596} C_DIS
LIN {X 69.1507,Y 93.2463,Z 126,A 49.4163,B 24.9361,C -1.8465,E1 25.0946,E2 396.4672} C_DIS
LIN {X 66.4222,Y 95.2067,Z 126,A 50.841,B 24.9366,C -1.8387,E1 25.0914,E2 395.066} C_DIS
LIN {X 64.0602,Y 96.8118,Z 126,A 52.4842,B 24.9357,C -1.8518,E1 25.0875,E2 393.3974} C_DIS
LIN {X 61.6082,Y 98.3903,Z 126,A 53.9009,B 24.9357,C -1.853,E1 25.0842,E2 391.9824} C_DIS
LIN {X 58.4542,Y 100.2986,Z 126,A 55.9002,B 24.9349,C -1.8639,E1 25.0793,E2 389.9634} C_DIS
LIN {X 54.7332,Y 102.3766,Z 126,A 57.9551,B 24.9349,C -1.8646,E1 25.0743,E2 387.9128} C_DIS
LIN {X 51.7582,Y 103.9102,Z 126,A 59.443,B 24.9352,C -1.8593,E1 25.0706,E2 386.4415} C_DIS
LIN {X 49.3885,Y 105.0579,Z 126,A 60.8871,B 24.9346,C -1.8675,E1 25.067,E2 384.9819} C_DIS
LIN {X 45.7431,Y 106.6971,Z 126,A 62.91,B 24.9343,C -1.8719,E1 25.0618,E2 382.9533} C_DIS
LIN {X 41.7807,Y 108.3101,Z 126,A 65.0164,B 24.9342,C -1.8738,E1 25.0563,E2 380.8472} C_DIS
LIN {X 38.4288,Y 109.5419,Z 126,A 66.6273,B 24.9345,C -1.8687,E1 25.0521,E2 379.2518} C_DIS
LIN {X 35.0683,Y 110.6657,Z 126,A 68.5181,B 24.934,C -1.8764,E1 25.0471,E2 377.3462} C_DIS
LIN {X 30.9972,Y 111.8742,Z 126,A 70.4364,B 24.9345,C -1.87,E1 25.042,E2 375.4465} C_DIS
LIN {X 28.2598,Y 112.5967,Z 126,A 71.9987,B 24.9339,C -1.8782,E1 25.0377,E2 373.8669} C_DIS
LIN {X 24.8821,Y 113.3892,Z 126,A 73.5418,B 24.9343,C -1.8716,E1 25.0335,E2 372.3416} C_DIS
LIN {X 20.7002,Y 114.2266,Z 126,A 75.3966,B 24.9351,C -1.8614,E1 25.0285,E2 370.5132} C_DIS
LIN {X 17.8965,Y 114.6993,Z 126,A 77.0629,B 24.9342,C -1.8735,E1 25.0239,E2 368.8199} C_DIS
LIN {X 14.8525,Y 115.133,Z 126,A 78.5124,B 24.9344,C -1.8709,E1 25.0199,E2 367.3778} C_DIS
LIN {X 11.3733,Y 115.5307,Z 126,A 80.2916,B 24.9342,C -1.8733,E1 25.0149,E2 365.594} C_DIS
LIN {X 7.9847,Y 115.8122,Z 126,A 81.722,B 24.935,C -1.8626,E1 25.011,E2 364.1899} C_DIS
LIN {X 5.1461,Y 115.973,Z 126,A 83.1682,B 24.9348,C -1.8644,E1 25.007,E2 362.7398} C_DIS
LIN {X 2.8613,Y 116.0539,Z 126,A 84.6787,B 24.9337,C -1.881,E1 25.0026,E2 361.1902} C_DIS
LIN {X -0.7487,Y 116.0846,Z 126,A 86.2392,B 24.9344,C -1.871,E1 24.9983,E2 359.6536} C_DIS
LIN {X -4.2697,Y 116.0106,Z 126,A 88.2028,B 24.9337,C -1.8803,E1 24.9928,E2 357.6676} C_DIS
LIN {X -7.1097,Y 115.8712,Z 126,A 89.6066,B 24.9337,C -1.8798,E1 24.9889,E2 356.2646} C_DIS
LIN {X -10.5457,Y 115.6071,Z 126,A 91.159,B 24.9343,C -1.8726,E1 24.9846,E2 354.7286} C_DIS
LIN {X -13.6573,Y 115.281,Z 126,A 92.7478,B 24.9342,C -1.8736,E1 24.9802,E2 353.1363} C_DIS
LIN {X -17.0286,Y 114.8334,Z 126,A 94.5364,B 24.9339,C -1.8773,E1 24.9752,E2 351.3376} C_DIS
LIN {X -19.8357,Y 114.382,Z 126,A 95.9408,B 24.934,C -1.8763,E1 24.9714,E2 349.9342} C_DIS
LIN {X -23.1245,Y 113.7607,Z 126,A 97.4208,B 24.9346,C -1.8675,E1 24.9674,E2 348.4733} C_DIS
LIN {X -26.0254,Y 113.1322,Z 126,A 98.8821,B 24.9347,C -1.8661,E1 24.9634,E2 347.0137} C_DIS
LIN {X -28.7573,Y 112.4688,Z 126,A 100.2729,B 24.9348,C -1.8648,E1 24.9596,E2 345.6238} C_DIS
LIN {X -32.2977,Y 111.5056,Z 126,A 102.0926,B 24.9349,C -1.8633,E1 24.9547,E2 343.8051} C_DIS
LIN {X -35.1505,Y 110.6391,Z 126,A 103.7126,B 24.9346,C -1.8679,E1 24.9504,E2 342.1711} C_DIS
LIN {X -39.0936,Y 109.3086,Z 126,A 105.8016,B 24.9346,C -1.8668,E1 24.9449,E2 340.0806} C_DIS
LIN {X -41.7505,Y 108.3215,Z 126,A 107.0304,B 24.9353,C -1.8577,E1 24.9417,E2 338.871} C_DIS
LIN {X -44.4227,Y 107.2535,Z 126,A 108.5893,B 24.935,C -1.8616,E1 24.9376,E2 337.2993} C_DIS
LIN {X -48.3392,Y 105.5463,Z 126,A 110.5707,B 24.9356,C -1.853,E1 24.9326,E2 335.3336} C_DIS
LIN {X -50.932,Y 104.3197,Z 126,A 112.1678,B 24.9353,C -1.8584,E1 24.9286,E2 333.7195} C_DIS
LIN {X -54.7247,Y 102.3812,Z 126,A 114.1011,B 24.936,C -1.8477,E1 24.9238,E2 331.8063} C_DIS
LIN {X -57.695,Y 100.7349,Z 126,A 115.5379,B 24.9369,C -1.8348,E1 24.9204,E2 330.3961} C_DIS
LIN {X -59.6659,Y 99.5824,Z 126,A 116.9153,B 24.9363,C -1.8432,E1 24.917,E2 328.9946} C_DIS
LIN {X -62.0825,Y 98.094,Z 126,A 118.3216,B 24.9365,C -1.8408,E1 24.9137,E2 327.5896} C_DIS
LIN {X -64.9514,Y 96.2161,Z 126,A 120.0622,B 24.9365,C -1.8395,E1 24.9096,E2 325.8463} C_DIS
LIN {X -67.8963,Y 94.1628,Z 126,A 121.8965,B 24.9366,C -1.8385,E1 24.9054,E2 324.0081} C_DIS
LIN {X -70.8785,Y 91.9371,Z 126,A 123.7452,B 24.9369,C -1.8351,E1 24.9013,E2 322.1608} C_DIS
LIN {X -74.0364,Y 89.4139,Z 126,A 125.7025,B 24.9373,C -1.8291,E1 24.8971,E2 320.2103} C_DIS
LIN {X -76.3706,Y 87.4284,Z 126,A 127.1696,B 24.9377,C -1.8238,E1 24.894,E2 318.7502} C_DIS
LIN {X -78.4869,Y 85.5336,Z 126,A 128.5788,B 24.9379,C -1.8208,E1 24.8911,E2 317.3424} C_DIS
LIN {X -80.5563,Y 83.5875,Z 126,A 129.9881,B 24.9381,C -1.8177,E1 24.8883,E2 315.9346} C_DIS
LIN {X -82.7116,Y 81.4556,Z 126,A 131.5592,B 24.9381,C -1.8172,E1 24.8852,E2 314.3581} C_DIS
LIN {X -85.3515,Y 78.6854,Z 126,A 133.3371,B 24.9387,C -1.8078,E1 24.8818,E2 312.5947} C_DIS
LIN {X -87.2511,Y 76.5736,Z 126,A 134.7463,B 24.939,C -1.8045,E1 24.8792,E2 311.1871} C_DIS
LIN {X -88.9999,Y 74.5346,Z 126,A 136.1336,B 24.939,C -1.8036,E1 24.8767,E2 309.7957} C_DIS
LIN {X -91.0223,Y 72.0495,Z 126,A 137.7485,B 24.9392,C -1.8008,E1 24.8738,E2 308.18} C_DIS
LIN {X -92.9121,Y 69.5958,Z 126,A 139.3333,B 24.9393,C -1.7989,E1 24.8712,E2 306.5919} C_DIS
LIN {X -94.9391,Y 66.8072,Z 126,A 140.9694,B 24.9398,C -1.7915,E1 24.8685,E2 304.9656} C_DIS
LIN {X -96.8405,Y 64.0166,Z 126,A 142.666,B 24.9401,C -1.7881,E1 24.8659,E2 303.2687} C_DIS
LIN {X -98.3703,Y 61.6402,Z 126,A 144.0523,B 24.9404,C -1.7837,E1 24.8638,E2 301.8857} C_DIS
LIN {X -100.2781,Y 58.4888,Z 126,A 146.0523,B 24.9402,C -1.7859,E1 24.8609,E2 299.8703} C_DIS
LIN {X -101.9288,Y 55.5588,Z 126,A 147.6254,B 24.9408,C -1.7775,E1 24.8588,E2 298.309} C_DIS
LIN {X -103.4398,Y 52.6919,Z 126,A 149.2357,B 24.9411,C -1.7731,E1 24.8567,E2 296.7003} C_DIS
LIN {X -105.175,Y 49.1369,Z 126,A 150.8837,B 24.9423,C -1.7548,E1 24.8548,E2 295.0872} C_DIS
LIN {X -106.3464,Y 46.5475,Z 126,A 152.5933,B 24.9417,C -1.763,E1 24.8528,E2 293.3486} C_DIS
LIN {X -107.4849,Y 43.8543,Z 126,A 153.9803,B 24.9422,C -1.7563,E1 24.8513,E2 291.9699} C_DIS
LIN {X -108.4022,Y 41.5376,Z 126,A 155.329,B 24.9422,C -1.7573,E1 24.85,E2 290.6113} C_DIS
LIN {X -109.7782,Y 37.755,Z 126,A 157.3655,B 24.9424,C -1.753,E1 24.8481,E2 288.5733} C_DIS
LIN {X -110.8344,Y 34.5247,Z 126,A 158.922,B 24.9431,C -1.7428,E1 24.8468,E2 287.0322} C_DIS
LIN {X -111.882,Y 30.9694,Z 126,A 160.768,B 24.9434,C -1.7376,E1 24.8453,E2 285.1879} C_DIS
LIN {X -112.6106,Y 28.2054,Z 126,A 162.1846,B 24.9437,C -1.7334,E1 24.8444,E2 283.7732} C_DIS
LIN {X -113.3853,Y 24.8997,Z 126,A 163.8788,B 24.944,C -1.7287,E1 24.8433,E2 282.0802} C_DIS
LIN {X -114.2262,Y 20.7028,Z 126,A 165.7506,B 24.9451,C -1.7121,E1 24.8423,E2 280.2369} C_DIS
LIN {X -114.6976,Y 17.9076,Z 126,A 167.1663,B 24.9453,C -1.7082,E1 24.8417,E2 278.8221} C_DIS
LIN {X -115.1004,Y 15.1038,Z 126,A 168.8146,B 24.945,C -1.7138,E1 24.841,E2 277.1505} C_DIS
LIN {X -115.4344,Y 12.2938,Z 126,A 170.2838,B 24.945,C -1.7122,E1 24.8406,E2 275.6764} C_DIS
LIN {X -115.7311,Y 9.0853,Z 126,A 171.8969,B 24.9453,C -1.708,E1 24.8402,E2 274.0637} C_DIS
LIN {X -115.9735,Y 5.1352,Z 126,A 173.5413,B 24.9465,C -1.689,E1 24.8399,E2 272.4546} C_DIS
LIN {X -116.0542,Y 2.8518,Z 126,A 174.9285,B 24.9461,C -1.6959,E1 24.8399,E2 271.0428} C_DIS
LIN {X -116.0865,Y -0.5181,Z 126,A 176.6533,B 24.9463,C -1.693,E1 24.8398,E2 269.3145} C_DIS
LIN {X -116.0101,Y -4.2822,Z 126,A 178.6531,B 24.9463,C -1.6927,E1 24.84,E2 267.3033} C_DIS
LIN {X -115.82,Y -7.869,Z 126,A -179.787,B 24.9472,C -1.6783,E1 24.8402,E2 265.7683} C_DIS
LIN {X -115.5304,Y -11.3764,Z 126,A -177.9728,B 24.9474,C -1.6758,E1 24.8407,E2 263.9492} C_DIS
LIN {X -115.1809,Y -14.4827,Z 126,A -176.3649,B 24.9475,C -1.6735,E1 24.8412,E2 262.3371} C_DIS
LIN {X -114.7173,Y -17.7805,Z 126,A -174.7082,B 24.9478,C -1.6688,E1 24.8419,E2 260.6818} C_DIS
LIN {X -114.1357,Y -21.206,Z 126,A -173.0666,B 24.9483,C -1.6603,E1 24.8427,E2 259.0506} C_DIS
LIN {X -113.5702,Y -24.0522,Z 126,A -171.4369,B 24.9481,C -1.6639,E1 24.8436,E2 257.4027} C_DIS
LIN {X -112.8181,Y -27.3551,Z 126,A -169.9329,B 24.9489,C -1.6519,E1 24.8446,E2 255.9187} C_DIS
LIN {X -111.8929,Y -30.9295,Z 126,A -168.0958,B 24.9492,C -1.6468,E1 24.8459,E2 254.083} C_DIS
LIN {X -110.9324,Y -34.2086,Z 126,A -166.3909,B 24.9495,C -1.6424,E1 24.8473,E2 252.3787} C_DIS
LIN {X -110.0522,Y -36.9422,Z 126,A -164.9724,B 24.9497,C -1.6382,E1 24.8485,E2 250.9622} C_DIS
LIN {X -108.6186,Y -40.966,Z 126,A -162.8191,B 24.95,C -1.6337,E1 24.8505,E2 248.8074} C_DIS
LIN {X -107.4614,Y -43.9122,Z 126,A -161.2071,B 24.9501,C -1.6312,E1 24.8522,E2 247.1924} C_DIS
LIN {X -105.8911,Y -47.574,Z 126,A -159.5457,B 24.9513,C -1.6129,E1 24.854,E2 245.5654} C_DIS
LIN {X -104.9379,Y -49.6461,Z 126,A -158.1681,B 24.9508,C -1.62,E1 24.8557,E2 244.1633} C_DIS
LIN {X -103.4402,Y -52.6909,Z 126,A -156.4823,B 24.9511,C -1.6158,E1 24.8578,E2 242.4785} C_DIS
LIN {X -101.7102,Y -55.9618,Z 126,A -154.4629,B 24.9509,C -1.6187,E1 24.8605,E2 240.4414} C_DIS
LIN {X -99.9103,Y -59.1112,Z 126,A -152.8216,B 24.9516,C -1.6077,E1 24.8628,E2 238.8179} C_DIS
LIN {X -98.0677,Y -62.1241,Z 126,A -151.0914,B 24.9519,C -1.6025,E1 24.8653,E2 237.0912} C_DIS
LIN {X -96.2066,Y -64.9654,Z 126,A -149.4046,B 24.9521,C -1.5986,E1 24.8679,E2 235.4052} C_DIS
LIN {X -94.5881,Y -67.3001,Z 126,A -147.9948,B 24.9523,C -1.5954,E1 24.8702,E2 233.9962} C_DIS
LIN {X -92.913,Y -69.5945,Z 126,A -146.5461,B 24.9524,C -1.5938,E1 24.8726,E2 232.5442} C_DIS
LIN {X -91.085,Y -71.9703,Z 126,A -145.0628,B 24.9526,C -1.5904,E1 24.8751,E2 231.0621} C_DIS
LIN {X -88.8271,Y -74.7425,Z 126,A -143.1724,B 24.9526,C -1.5915,E1 24.8785,E2 229.1604} C_DIS
LIN {X -86.7794,Y -77.1084,Z 126,A -141.6836,B 24.9529,C -1.5856,E1 24.8813,E2 227.6789} C_DIS
LIN {X -84.5718,Y -79.5223,Z 126,A -140.1461,B 24.9533,C -1.5788,E1 24.8842,E2 226.1509} C_DIS
LIN {X -82.5885,Y -81.5802,Z 126,A -138.7079,B 24.9534,C -1.5768,E1 24.887,E2 224.7111} C_DIS
LIN {X -80.2506,Y -83.8822,Z 126,A -136.9359,B 24.9532,C -1.5799,E1 24.8906,E2 222.9245} C_DIS
LIN {X -77.4985,Y -86.4303,Z 126,A -135.2238,B 24.9538,C -1.5702,E1 24.8941,E2 221.2284} C_DIS
LIN {X -75.2874,Y -88.3629,Z 126,A -133.7903,B 24.954,C -1.5667,E1 24.8971,E2 219.7977} C_DIS
LIN {X -73.0863,Y -90.1919,Z 126,A -132.3723,B 24.9542,C -1.5643,E1 24.9002,E2 218.3802} C_DIS
LIN {X -70.8577,Y -91.9531,Z 126,A -130.9338,B 24.9542,C -1.5633,E1 24.9033,E2 216.9387} C_DIS
LIN {X -68.0162,Y -94.077,Z 126,A -129.2062,B 24.9545,C -1.5592,E1 24.9072,E2 215.2148} C_DIS
LIN {X -65.6788,Y -95.7235,Z 126,A -127.6112,B 24.9541,C -1.5647,E1 24.9109,E2 213.6012} C_DIS
LIN {X -62.8372,Y -97.61,Z 126,A -126.0998,B 24.9547,C -1.5547,E1 24.9144,E2 212.1088} C_DIS
LIN {X -60.4227,Y -99.1228,Z 126,A -124.6908,B 24.9548,C -1.5527,E1 24.9177,E2 210.7002} C_DIS
LIN {X -56.7225,Y -101.2856,Z 126,A -122.573,B 24.955,C -1.5497,E1 24.9229,E2 208.583} C_DIS
LIN {X -54.5028,Y -102.4981,Z 126,A -121.4279,B 24.9554,C -1.5436,E1 24.9257,E2 207.4493} C_DIS
LIN {X -51.7589,Y -103.9099,Z 126,A -119.7984,B 24.9552,C -1.5462,E1 24.9297,E2 205.8091} C_DIS
LIN {X -49.132,Y -105.1773,Z 126,A -118.303,B 24.9552,C -1.547,E1 24.9335,E2 204.3082} C_DIS
LIN {X -46.5363,Y -106.3513,Z 126,A -117.0619,B 24.9557,C -1.5382,E1 24.9366,E2 203.0849} C_DIS
LIN {X -43.9108,Y -107.4619,Z 126,A -115.5267,B 24.9554,C -1.5423,E1 24.9406,E2 201.5364} C_DIS
LIN {X -41.501,Y -108.416,Z 126,A -114.1656,B 24.9553,C -1.5447,E1 24.9442,E2 200.1669} C_DIS
LIN {X -37.7749,Y -109.7713,Z 126,A -112.2831,B 24.9556,C -1.5397,E1 24.9491,E2 198.2925} C_DIS
LIN {X -34.557,Y -110.8244,Z 126,A -110.6123,B 24.9556,C -1.5384,E1 24.9536,E2 196.6217} C_DIS
LIN {X -31.8488,Y -111.6328,Z 126,A -109.1541,B 24.9556,C -1.5402,E1 24.9575,E2 195.1569} C_DIS
LIN {X -28.6211,Y -112.5038,Z 126,A -107.5127,B 24.9556,C -1.5388,E1 24.9619,E2 193.5164} C_DIS
LIN {X -24.8867,Y -113.3882,Z 126,A -105.6645,B 24.9558,C -1.5358,E1 24.967,E2 191.6728} C_DIS
LIN {X -20.7048,Y -114.2258,Z 126,A -103.5105,B 24.9558,C -1.5372,E1 24.9729,E2 189.5132} C_DIS
LIN {X -17.523,Y -114.7571,Z 126,A -101.907,B 24.9558,C -1.5372,E1 24.9773,E2 187.9081} C_DIS
LIN {X -13.6515,Y -115.2816,Z 126,A -100.0355,B 24.9558,C -1.5343,E1 24.9825,E2 186.0422} C_DIS
LIN {X -9.9642,Y -115.6608,Z 126,A -98.0276,B 24.9554,C -1.5421,E1 24.9881,E2 184.0148} C_DIS
LIN {X -7.1296,Y -115.87,Z 126,A -96.6262,B 24.9554,C -1.5421,E1 24.992,E2 182.613} C_DIS
LIN {X -4.2913,Y -116.0097,Z 126,A -95.3994,B 24.9559,C -1.5343,E1 24.9954,E2 181.4043} C_DIS
LIN {X -0.865,Y -116.0839,Z 126,A -93.9583,B 24.9565,C -1.5235,E1 24.9993,E2 179.9889} C_DIS
LIN {X 0.8095,Y -116.0815,Z 126,A -93.0664,B 24.9563,C -1.5266,E1 25.0019,E2 179.0896} C_DIS
Enddeposition()
LIN {X 0.8647,Y -121.7874,Z 127,A -92.827,B 24.9609,C -1.4452,E1 25.0019,E2 179.043} C_DIS
Startdeposition()
$VEL.CP = VEL_PRINT
LIN {X -2.989,Y -121.7576,Z 127,A -95.1241,B 24.9621,C -1.422,E1 24.9954,E2 181.3953} C_DIS
LIN {X -5.9762,Y -121.6476,Z 127,A -96.5302,B 24.9621,C -1.4218,E1 24.9915,E2 182.802} C_DIS
LIN {X -8.9597,Y -121.4643,Z 127,A -97.9363,B 24.9621,C -1.4218,E1 24.9876,E2 184.2086} C_DIS
LIN {X -11.6165,Y -121.2375,Z 127,A -99.2098,B 24.9621,C -1.421,E1 24.984,E2 185.4847} C_DIS
LIN {X -14.387,Y -120.9395,Z 127,A -100.5023,B 24.9621,C -1.4221,E1 24.9804,E2 186.7754} C_DIS
LIN {X -17.8709,Y -120.4761,Z 127,A -102.1562,B 24.9621,C -1.4224,E1 24.9759,E2 188.4299} C_DIS
LIN {X -20.8222,Y -120.0012,Z 127,A -103.5636,B 24.9621,C -1.4228,E1 24.972,E2 189.8378} C_DIS
LIN {X -23.7609,Y -119.4541,Z 127,A -104.971,B 24.9621,C -1.4233,E1 24.9681,E2 191.2456} C_DIS
LIN {X -26.6853,Y -118.835,Z 127,A -106.3787,B 24.9621,C -1.4239,E1 24.9643,E2 192.6536} C_DIS
LIN {X -29.5936,Y -118.1443,Z 127,A -107.7865,B 24.962,C -1.4246,E1 24.9605,E2 194.0616} C_DIS
LIN {X -33.4165,Y -117.1182,Z 127,A -109.6513,B 24.962,C -1.4257,E1 24.9554,E2 195.9267} C_DIS
LIN {X -36.2807,Y -116.2629,Z 127,A -111.0596,B 24.9619,C -1.4266,E1 24.9517,E2 197.3353} C_DIS
LIN {X -39.6209,Y -115.1696,Z 127,A -112.7159,B 24.9619,C -1.4278,E1 24.9473,E2 198.9918} C_DIS
LIN {X -43.3418,Y -113.8193,Z 127,A -114.6398,B 24.9619,C -1.4267,E1 24.9422,E2 200.9222} C_DIS
LIN {X -47.5018,Y -112.1469,Z 127,A -116.6959,B 24.9616,C -1.4313,E1 24.9369,E2 202.9721} C_DIS
LIN {X -50.7188,Y -110.7315,Z 127,A -118.3532,B 24.9616,C -1.4329,E1 24.9327,E2 204.6295} C_DIS
LIN {X -52.9473,Y -109.681,Z 127,A -119.5153,B 24.9615,C -1.4342,E1 24.9298,E2 205.7914} C_DIS
LIN {X -55.6231,Y -108.3486,Z 127,A -120.9834,B 24.9615,C -1.4332,E1 24.9261,E2 207.2659} C_DIS
LIN {X -58.2653,Y -106.9509,Z 127,A -122.3871,B 24.9615,C -1.4352,E1 24.9227,E2 208.6687} C_DIS
LIN {X -61.3281,Y -105.227,Z 127,A -123.9941,B 24.9612,C -1.4396,E1 24.9188,E2 210.27} C_DIS
LIN {X -63.892,Y -103.6902,Z 127,A -125.405,B 24.9611,C -1.4415,E1 24.9154,E2 211.6807} C_DIS
LIN {X -66.4175,Y -102.091,Z 127,A -126.8158,B 24.961,C -1.4435,E1 24.9121,E2 213.0914} C_DIS
LIN {X -70.1302,Y -99.5772,Z 127,A -128.933,B 24.9608,C -1.4467,E1 24.9072,E2 215.2082} C_DIS
LIN {X -73.3277,Y -97.244,Z 127,A -130.8371,B 24.9608,C -1.4481,E1 24.9029,E2 217.1156} C_DIS
LIN {X -76.1043,Y -95.0893,Z 127,A -132.4618,B 24.9605,C -1.4524,E1 24.8994,E2 218.7361} C_DIS
LIN {X -78.415,Y -93.193,Z 127,A -133.8738,B 24.9603,C -1.4549,E1 24.8963,E2 220.1477} C_DIS
LIN {X -81.4255,Y -90.5718,Z 127,A -135.755,B 24.9602,C -1.4585,E1 24.8924,E2 222.0277} C_DIS
LIN {X -83.9821,Y -88.2092,Z 127,A -137.4046,B 24.96,C -1.4613,E1 24.889,E2 223.6774} C_DIS
LIN {X -87.1719,Y -85.0583,Z 127,A -139.5239,B 24.9598,C -1.4654,E1 24.8849,E2 225.7959} C_DIS
LIN {X -88.8731,Y -83.2761,Z 127,A -140.7467,B 24.9598,C -1.4652,E1 24.8825,E2 227.0245} C_DIS
LIN {X -91.8886,Y -79.9364,Z 127,A -142.8711,B 24.9595,C -1.4697,E1 24.8786,E2 229.1476} C_DIS
LIN {X -94.7585,Y -76.5126,Z 127,A -144.9284,B 24.9592,C -1.4767,E1 24.8749,E2 231.1979} C_DIS
LIN {X -96.6077,Y -74.164,Z 127,A -146.4003,B 24.9592,C -1.4772,E1 24.8724,E2 232.6754} C_DIS
LIN {X -98.7091,Y -71.3468,Z 127,A -148.0041,B 24.9588,C -1.4835,E1 24.8697,E2 234.2721} C_DIS
LIN {X -101.2683,Y -67.6653,Z 127,A -150.1252,B 24.9585,C -1.4884,E1 24.8664,E2 236.392} C_DIS
LIN {X -103.4118,Y -64.3377,Z 127,A -151.9981,B 24.9582,C -1.4929,E1 24.8636,E2 238.2637} C_DIS
LIN {X -104.9596,Y -61.7805,Z 127,A -153.4124,B 24.9581,C -1.4963,E1 24.8616,E2 239.6772} C_DIS
LIN {X -106.4442,Y -59.186,Z 127,A -154.8852,B 24.9581,C -1.4972,E1 24.8595,E2 241.1554} C_DIS
LIN {X -107.8646,Y -56.5559,Z 127,A -156.2998,B 24.9578,C -1.5008,E1 24.8577,E2 242.569} C_DIS
LIN {X -109.4534,Y -53.421,Z 127,A -157.9048,B 24.9574,C -1.5075,E1 24.8557,E2 244.1667} C_DIS
LIN {X -110.5097,Y -51.1951,Z 127,A -159.0712,B 24.9573,C -1.5106,E1 24.8543,E2 245.3322} C_DIS
LIN {X -111.9428,Y -47.986,Z 127,A -160.735,B 24.957,C -1.5149,E1 24.8524,E2 246.9948} C_DIS
LIN {X -113.0868,Y -45.2243,Z 127,A -162.15,B 24.9568,C -1.5186,E1 24.8509,E2 248.4088} C_DIS
LIN {X -114.1626,Y -42.4354,Z 127,A -163.5653,B 24.9566,C -1.5224,E1 24.8495,E2 249.823} C_DIS
LIN {X -114.9956,Y -40.1168,Z 127,A -164.7319,B 24.9564,C -1.5256,E1 24.8485,E2 250.9886} C_DIS
LIN {X -116.0177,Y -37.0593,Z 127,A -166.2785,B 24.9562,C -1.5289,E1 24.8471,E2 252.5362} C_DIS
LIN {X -116.975,Y -33.9221,Z 127,A -167.8115,B 24.9559,C -1.5341,E1 24.8459,E2 254.0658} C_DIS
LIN {X -117.7722,Y -31.0412,Z 127,A -169.2272,B 24.9557,C -1.538,E1 24.8449,E2 255.4803} C_DIS
LIN {X -118.374,Y -28.6521,Z 127,A -170.4524,B 24.9557,C -1.5388,E1 24.844,E2 256.7108} C_DIS
LIN {X -119.3484,Y -24.2756,Z 127,A -172.5179,B 24.9551,C -1.5473,E1 24.8428,E2 258.7681} C_DIS
LIN {X -120.0012,Y -20.8222,Z 127,A -174.1824,B 24.9549,C -1.5521,E1 24.842,E2 260.4313} C_DIS
Enddeposition()
END
